// TwinCAT 3 PLC project MasterArmControl
// ProgramVersion: 3.1.4024.0
// libraries:
//   Tc2_Math, * (Beckhoff Automation GmbH)
//   Tc2_Standard, * (Beckhoff Automation GmbH)
//   Tc2_System, * (Beckhoff Automation GmbH)
//   Tc2_Utilities, * (Beckhoff Automation GmbH)
//   Tc3_Module, * (Beckhoff Automation GmbH)
// project tree:
//   AgiMaths/ DHTrans.TcPOU, sign.TcPOU, addVec7.TcPOU (not stored), multiNumVec3.TcPOU, multiNumVec7.TcPOU, normVec3.TcPOU, normVec7.TcPOU, subVec7.TcPOU (not stored), subVec3.TcPOU (not stored), addVec3.TcPOU (not stored), atan2.TcPOU (not stored), cot.TcPOU (not stored), mat3Mat3.TcPOU (not stored), mat3Vec3.TcPOU (not stored), mat67Vec7.TcPOU (not stored), rotZ.TcPOU (not stored), rotY.TcPOU (not stored), rotX.TcPOU (not stored), transform.TcPOU (not stored)
//   DUTs/Structure/Communication/ ST_MasterDynaData.TcDUT, ST_UIData.TcDUT, ST_CartStatus.TcDUT, ST_MasterStatus.TcDUT, ST_MasterJointData.TcDUT, ST_MotorInputs.TcDUT (not stored), ST_MotorOutputs.TcDUT (not stored), ST_SlaveStatus.TcDUT, ST_SlaveJointData.TcDUT, ST_SafetyData.TcDUT (not stored)
//   DUTs/Structure/ ST_ArmCtrlCmds.TcDUT, ST_MasterInputDataPool.TcDUT, ST_Frame.TcDUT, ST_InstruStatus.TcDUT
//   DUTs/Type/ Mat37.TcDUT (not stored), Mat4d.TcDUT (not stored), Mat5d.TcDUT (not stored), Mat67.TcDUT, Mat6d.TcDUT, Mat76.TcDUT, Mat7d.TcDUT, Vec4d.TcDUT (not stored), Mat3d.TcDUT, Vec3d.TcDUT, Vec6d.TcDUT, Vec7d.TcDUT (not stored), Vec7i.TcDUT (not stored)
//   FBs_BasicControllers/ FB_RedunJntControl.TcPOU (not stored), FB_PID.TcPOU
//   DUTs/Enum/ E_DriverCtrlWord.TcDUT (not stored), E_DriverOPMode.TcDUT (not stored), E_DriverStatusWord.TcDUT, E_InstrumentType.TcDUT (not stored), E_MasterArmState.TcDUT (not stored), E_MatchedSlaveArmIdx.TcDUT (not stored), E_SlaveArmState.TcDUT
//   FBs_RobotDynamics/ FB_MasterDynamic.TcPOU, FB_MasterGravity.TcPOU
//   FBs_StateControllers/ FB_ArmClutch.TcPOU, FB_ArmEndoscope.TcPOU, FB_ArmCart.TcPOU, FB_ArmMatching.TcPOU, FB_ArmHome.TcPOU, FB_ArmError.TcPOU, FB_ArmReady.TcPOU, FB_ArmMasterSlave.TcPOU, FB_ArmInit.TcPOU, FB_ArmStandBy.TcPOU, FB_MasterArmCtrlBase.TcPOU, I_MasterArmCtrl.TcIO
//   FBs_TrajectoryPlanning/ FB_BasicDoubleS.TcPOU, FB_trajBase.TcPOU (not stored), FB_TrajMoveJ.TcPOU, linear_trajectory_with_quintic_polynomial_blends.TcPOU, quintic_spline_curve.TcPOU, Quintic_spline_curve_factor.TcPOU, TrapezoIDal_velocity_trajectory.TcPOU
//   FBs_TrajectoryPlanning/OTG/ FB_secOrdTrajFilter.TcPOU (not stored), FB_thirdOrdTrajFilter.TcPOU
//   FBs_Filters/ FB_LowPassFilter.TcPOU (not stored)
//   GVLs/ GVLs_ArmDynamics.TcGVL (not stored), GVL_ArmKinematic.TcGVL (not stored), GVL_CartParameters.TcGVL (not stored), GVL_ControlParameters.TcGVL, GVL_JointEncoderCaliData.TcGVL, GVL_MathDefine.TcGVL, GVL_MotorParameters.TcGVL, GVL_SafetyParameters.TcGVL (not stored), GVL_SystemParameters.TcGVL
//   FBs_Robots/ FB_Joint.TcPOU, FB_MasterArm.TcPOU, FB_MasterRobot.TcPOU
//   MatrixLib/ cross.TcPOU, Det5.TcPOU, Det6.TcPOU, Det7.TcPOU, invMat6Old.TcPOU, invMat7.TcPOU, invMat6.TcPOU, Mat3T.TcPOU, vecSelfMultiNum.TcPOU, matMultiVec.TcPOU, matMultiply.TcPOU, matMultiNum.TcPOU, matSelfSub.TcPOU, matAdd.TcPOU, matSelfAdd.TcPOU (not stored), matTranspose.TcPOU, matSub.TcPOU (not stored)
//   / TaskArmControl.TcTTO, TaskDynamic.TcTTO
//   Mains/ MasterArmControl.TcPOU, RobotDynamics.TcPOU
// real-time tasks:
//   TASK TaskArmControl: cycle T#1ms, priority 20, ADS port 350
//   TASK TaskDynamic: cycle T#1ms, priority 1, ADS port 351
// I/O:
//   DEVICE Device 3 (EtherCAT) (disabled), AmsNetId 169.254.206.98.4.1
//     Box 26 (AX58200_MotorControl) [AX58200_MotorControl2021.9.13]
//     Box 27 (EL6695-0002) [EL6695 EtherCAT Bridge terminal (Secondary)]
//   DEVICE LeftArm (EtherCAT), AmsNetId 169.254.206.98.3.1
//     Joint1 (AX58200_MotorControl) [AX58200_MotorControl_1axis]
//     Joint2 (AX58200_MotorControl) [AX58200_MotorControl_1axis]
//     Joint3 (AX58200_MotorControl) [AX58200_MotorControl_1axis]
//     Joint4 (AX58200_MotorControl) [AX58200_MotorControl_1axis]
//     Joint5 (AX58200_MotorControl) [AX58200_MotorControl_1axis]
//     Joint6 (AX58200_MotorControl) [AX58200_MotorControl_1axis]
//     Joint7 (AX58200_MotorControl) [AX58200_MotorControl_1axis]
//   DEVICE RightArm (EtherCAT), AmsNetId 169.254.206.98.7.1
//     Term 1 (EK1100) [EK1100 EtherCAT Coupler (2A E-Bus)]
//       Term 2 (EL6070) [EL6070 1Ch. Licensing-Terminal]
//       Term 3 (EL1008) [EL1008 8Ch. Dig. Input 24V, 3ms]
//       Term 4 (EL1008) [EL1008 8Ch. Dig. Input 24V, 3ms]
//       Term 5 (EL1008) [EL1008 8Ch. Dig. Input 24V, 3ms]
//       Term 6 (EL2008-0015) [EL2008-0015 8K. Dig. Ausgang 24V DC, 0.35A, nicht kurzschlussfest]
//       Term 7 (EK1122) [EK1122 2 port EtherCAT junction]
//         Box 8 (AX58200_MotorControl) [AX58200_MotorControl_1axis]
//         Box 9 (AX58200_MotorControl) [AX58200_MotorControl_1axis]
//         Box 10 (AX58200_MotorControl) [AX58200_MotorControl_1axis]
//         Box 11 (AX58200_MotorControl) [AX58200_MotorControl_1axis]
//     Joint1 (AX58200_MotorControl) [AX58200_MotorControl_1axis]
//     Joint2 (AX58200_MotorControl) [AX58200_MotorControl_1axis]
//     Joint3 (AX58200_MotorControl) [AX58200_MotorControl_1axis]
//     Joint4 (AX58200_MotorControl) [AX58200_MotorControl_1axis]
//     Joint5 (AX58200_MotorControl) [AX58200_MotorControl_1axis]
//     Joint6 (AX58200_MotorControl) [AX58200_MotorControl_1axis]
//     Joint7 (AX58200_MotorControl) [AX58200_MotorControl_1axis]
// variable links:
//   MasterArmControl/MasterArmControl Instance <-> LeftArm (EtherCAT)/Joint1 (AX58200_MotorControl)
//     TaskArmControl Inputs/MasterArmControl.m_masterRobot.m_masterArms[1].m_joints[1].m_motorInputs/m_current <-> TxPdoMappingCspCsv/Torque actual value
//     TaskArmControl Inputs/MasterArmControl.m_masterRobot.m_masterArms[1].m_joints[1].m_motorInputs/m_driverError <-> TxPdoMappingCspCsv/digital input
//     TaskArmControl Inputs/MasterArmControl.m_masterRobot.m_masterArms[1].m_joints[1].m_motorInputs/m_linkEncoder <-> TxPdoMappingCspCsv/ENC2
//     TaskArmControl Inputs/MasterArmControl.m_masterRobot.m_masterArms[1].m_joints[1].m_motorInputs/m_motorEncoder <-> TxPdoMappingCspCsv/Position actual value
//     TaskArmControl Inputs/MasterArmControl.m_masterRobot.m_masterArms[1].m_joints[1].m_motorInputs/m_statusWord <-> TxPdoMappingCspCsv/Statusword
//     TaskArmControl Outputs/MasterArmControl.m_masterRobot.m_masterArms[1].m_joints[1].m_motorOutputs/m_cmdCurrent <-> RxPdoMappingCspCsv/Target torque
//     TaskArmControl Outputs/MasterArmControl.m_masterRobot.m_masterArms[1].m_joints[1].m_motorOutputs/m_cmdMotorEncoder <-> RxPdoMappingCspCsv/Target position
//     TaskArmControl Outputs/MasterArmControl.m_masterRobot.m_masterArms[1].m_joints[1].m_motorOutputs/m_controlWord <-> RxPdoMappingCspCsv/Controlword
//     TaskArmControl Outputs/MasterArmControl.m_masterRobot.m_masterArms[1].m_joints[1].m_motorOutputs/m_opMode <-> RxPdoMappingCspCsv/Modes of operation
//   MasterArmControl/MasterArmControl Instance <-> LeftArm (EtherCAT)/Joint2 (AX58200_MotorControl)
//     TaskArmControl Inputs/MasterArmControl.m_masterRobot.m_masterArms[1].m_joints[2].m_motorInputs/m_current <-> TxPdoMappingCspCsv/Torque actual value
//     TaskArmControl Inputs/MasterArmControl.m_masterRobot.m_masterArms[1].m_joints[2].m_motorInputs/m_driverError <-> TxPdoMappingCspCsv/digital input
//     TaskArmControl Inputs/MasterArmControl.m_masterRobot.m_masterArms[1].m_joints[2].m_motorInputs/m_linkEncoder <-> TxPdoMappingCspCsv/ENC2
//     TaskArmControl Inputs/MasterArmControl.m_masterRobot.m_masterArms[1].m_joints[2].m_motorInputs/m_motorEncoder <-> TxPdoMappingCspCsv/Position actual value
//     TaskArmControl Inputs/MasterArmControl.m_masterRobot.m_masterArms[1].m_joints[2].m_motorInputs/m_statusWord <-> TxPdoMappingCspCsv/Statusword
//     TaskArmControl Outputs/MasterArmControl.m_masterRobot.m_masterArms[1].m_joints[2].m_motorOutputs/m_cmdCurrent <-> RxPdoMappingCspCsv/Target torque
//     TaskArmControl Outputs/MasterArmControl.m_masterRobot.m_masterArms[1].m_joints[2].m_motorOutputs/m_cmdMotorEncoder <-> RxPdoMappingCspCsv/Target position
//     TaskArmControl Outputs/MasterArmControl.m_masterRobot.m_masterArms[1].m_joints[2].m_motorOutputs/m_controlWord <-> RxPdoMappingCspCsv/Controlword
//     TaskArmControl Outputs/MasterArmControl.m_masterRobot.m_masterArms[1].m_joints[2].m_motorOutputs/m_opMode <-> RxPdoMappingCspCsv/Modes of operation
//   MasterArmControl/MasterArmControl Instance <-> LeftArm (EtherCAT)/Joint3 (AX58200_MotorControl)
//     TaskArmControl Inputs/MasterArmControl.m_masterRobot.m_masterArms[1].m_joints[3].m_motorInputs/m_current <-> TxPdoMappingCspCsv/Torque actual value
//     TaskArmControl Inputs/MasterArmControl.m_masterRobot.m_masterArms[1].m_joints[3].m_motorInputs/m_driverError <-> TxPdoMappingCspCsv/digital input
//     TaskArmControl Inputs/MasterArmControl.m_masterRobot.m_masterArms[1].m_joints[3].m_motorInputs/m_linkEncoder <-> TxPdoMappingCspCsv/ENC2
//     TaskArmControl Inputs/MasterArmControl.m_masterRobot.m_masterArms[1].m_joints[3].m_motorInputs/m_motorEncoder <-> TxPdoMappingCspCsv/Position actual value
//     TaskArmControl Inputs/MasterArmControl.m_masterRobot.m_masterArms[1].m_joints[3].m_motorInputs/m_statusWord <-> TxPdoMappingCspCsv/Statusword
//     TaskArmControl Outputs/MasterArmControl.m_masterRobot.m_masterArms[1].m_joints[3].m_motorOutputs/m_cmdCurrent <-> RxPdoMappingCspCsv/Target torque
//     TaskArmControl Outputs/MasterArmControl.m_masterRobot.m_masterArms[1].m_joints[3].m_motorOutputs/m_cmdMotorEncoder <-> RxPdoMappingCspCsv/Target position
//     TaskArmControl Outputs/MasterArmControl.m_masterRobot.m_masterArms[1].m_joints[3].m_motorOutputs/m_controlWord <-> RxPdoMappingCspCsv/Controlword
//     TaskArmControl Outputs/MasterArmControl.m_masterRobot.m_masterArms[1].m_joints[3].m_motorOutputs/m_opMode <-> RxPdoMappingCspCsv/Modes of operation
//   MasterArmControl/MasterArmControl Instance <-> LeftArm (EtherCAT)/Joint4 (AX58200_MotorControl)
//     TaskArmControl Inputs/MasterArmControl.m_masterRobot.m_masterArms[1].m_joints[4].m_motorInputs/m_current <-> TxPdoMappingCspCsv/Torque actual value
//     TaskArmControl Inputs/MasterArmControl.m_masterRobot.m_masterArms[1].m_joints[4].m_motorInputs/m_driverError <-> TxPdoMappingCspCsv/digital input
//     TaskArmControl Inputs/MasterArmControl.m_masterRobot.m_masterArms[1].m_joints[4].m_motorInputs/m_motorEncoder <-> TxPdoMappingCspCsv/Position actual value
//     TaskArmControl Inputs/MasterArmControl.m_masterRobot.m_masterArms[1].m_joints[4].m_motorInputs/m_statusWord <-> TxPdoMappingCspCsv/Statusword
//     TaskArmControl Outputs/MasterArmControl.m_masterRobot.m_masterArms[1].m_joints[4].m_motorOutputs/m_cmdCurrent <-> RxPdoMappingCspCsv/Target torque
//     TaskArmControl Outputs/MasterArmControl.m_masterRobot.m_masterArms[1].m_joints[4].m_motorOutputs/m_cmdMotorEncoder <-> RxPdoMappingCspCsv/Target position
//     TaskArmControl Outputs/MasterArmControl.m_masterRobot.m_masterArms[1].m_joints[4].m_motorOutputs/m_controlWord <-> RxPdoMappingCspCsv/Controlword
//     TaskArmControl Outputs/MasterArmControl.m_masterRobot.m_masterArms[1].m_joints[4].m_motorOutputs/m_opMode <-> RxPdoMappingCspCsv/Modes of operation
//   MasterArmControl/MasterArmControl Instance <-> LeftArm (EtherCAT)/Joint5 (AX58200_MotorControl)
//     TaskArmControl Inputs/MasterArmControl.m_masterRobot.m_masterArms[1].m_joints[4].m_motorInputs/m_linkEncoder <-> TxPdoMappingCspCsv/Velocity actual value
//     TaskArmControl Inputs/MasterArmControl.m_masterRobot.m_masterArms[1].m_joints[5].m_motorInputs/m_current <-> TxPdoMappingCspCsv/Torque actual value
//     TaskArmControl Inputs/MasterArmControl.m_masterRobot.m_masterArms[1].m_joints[5].m_motorInputs/m_driverError <-> TxPdoMappingCspCsv/digital input
//     TaskArmControl Inputs/MasterArmControl.m_masterRobot.m_masterArms[1].m_joints[5].m_motorInputs/m_linkEncoder <-> TxPdoMappingCspCsv/ENC2
//     TaskArmControl Inputs/MasterArmControl.m_masterRobot.m_masterArms[1].m_joints[5].m_motorInputs/m_motorEncoder <-> TxPdoMappingCspCsv/Position actual value
//     TaskArmControl Inputs/MasterArmControl.m_masterRobot.m_masterArms[1].m_joints[5].m_motorInputs/m_statusWord <-> TxPdoMappingCspCsv/Statusword
//     TaskArmControl Outputs/MasterArmControl.m_masterRobot.m_masterArms[1].m_joints[5].m_motorOutputs/m_cmdCurrent <-> RxPdoMappingCspCsv/Target torque
//     TaskArmControl Outputs/MasterArmControl.m_masterRobot.m_masterArms[1].m_joints[5].m_motorOutputs/m_cmdMotorEncoder <-> RxPdoMappingCspCsv/Target position
//     TaskArmControl Outputs/MasterArmControl.m_masterRobot.m_masterArms[1].m_joints[5].m_motorOutputs/m_controlWord <-> RxPdoMappingCspCsv/Controlword
//     TaskArmControl Outputs/MasterArmControl.m_masterRobot.m_masterArms[1].m_joints[5].m_motorOutputs/m_opMode <-> RxPdoMappingCspCsv/Modes of operation
//   MasterArmControl/MasterArmControl Instance <-> LeftArm (EtherCAT)/Joint6 (AX58200_MotorControl)
//     TaskArmControl Inputs/MasterArmControl.m_masterRobot.m_masterArms[1].m_joints[6].m_motorInputs/m_current <-> TxPdoMappingCspCsv/Torque actual value
//     TaskArmControl Inputs/MasterArmControl.m_masterRobot.m_masterArms[1].m_joints[6].m_motorInputs/m_driverError <-> TxPdoMappingCspCsv/digital input
//     TaskArmControl Inputs/MasterArmControl.m_masterRobot.m_masterArms[1].m_joints[6].m_motorInputs/m_linkEncoder <-> TxPdoMappingCspCsv/ENC2
//     TaskArmControl Inputs/MasterArmControl.m_masterRobot.m_masterArms[1].m_joints[6].m_motorInputs/m_motorEncoder <-> TxPdoMappingCspCsv/Position actual value
//     TaskArmControl Inputs/MasterArmControl.m_masterRobot.m_masterArms[1].m_joints[6].m_motorInputs/m_statusWord <-> TxPdoMappingCspCsv/Statusword
//     TaskArmControl Outputs/MasterArmControl.m_masterRobot.m_masterArms[1].m_joints[6].m_motorOutputs/m_cmdCurrent <-> RxPdoMappingCspCsv/Target torque
//     TaskArmControl Outputs/MasterArmControl.m_masterRobot.m_masterArms[1].m_joints[6].m_motorOutputs/m_cmdMotorEncoder <-> RxPdoMappingCspCsv/Target position
//     TaskArmControl Outputs/MasterArmControl.m_masterRobot.m_masterArms[1].m_joints[6].m_motorOutputs/m_controlWord <-> RxPdoMappingCspCsv/Controlword
//     TaskArmControl Outputs/MasterArmControl.m_masterRobot.m_masterArms[1].m_joints[6].m_motorOutputs/m_opMode <-> RxPdoMappingCspCsv/Modes of operation
//   MasterArmControl/MasterArmControl Instance <-> LeftArm (EtherCAT)/Joint7 (AX58200_MotorControl)
//     TaskArmControl Inputs/MasterArmControl.m_masterRobot.m_masterArms[1].m_gripHallSensorValue <-> TxPdoMappingCspCsv/analog input
//     TaskArmControl Inputs/MasterArmControl.m_masterRobot.m_masterArms[1].m_joints[7].m_motorInputs/m_current <-> TxPdoMappingCspCsv/Torque actual value
//     TaskArmControl Inputs/MasterArmControl.m_masterRobot.m_masterArms[1].m_joints[7].m_motorInputs/m_driverError <-> TxPdoMappingCspCsv/digital input
//     TaskArmControl Inputs/MasterArmControl.m_masterRobot.m_masterArms[1].m_joints[7].m_motorInputs/m_linkEncoder <-> TxPdoMappingCspCsv/ENC2
//     TaskArmControl Inputs/MasterArmControl.m_masterRobot.m_masterArms[1].m_joints[7].m_motorInputs/m_motorEncoder <-> TxPdoMappingCspCsv/Position actual value
//     TaskArmControl Inputs/MasterArmControl.m_masterRobot.m_masterArms[1].m_joints[7].m_motorInputs/m_statusWord <-> TxPdoMappingCspCsv/Statusword
//     TaskArmControl Outputs/MasterArmControl.m_masterRobot.m_masterArms[1].m_joints[7].m_motorOutputs/m_cmdCurrent <-> RxPdoMappingCspCsv/Target torque
//     TaskArmControl Outputs/MasterArmControl.m_masterRobot.m_masterArms[1].m_joints[7].m_motorOutputs/m_cmdMotorEncoder <-> RxPdoMappingCspCsv/Target position
//     TaskArmControl Outputs/MasterArmControl.m_masterRobot.m_masterArms[1].m_joints[7].m_motorOutputs/m_controlWord <-> RxPdoMappingCspCsv/Controlword
//     TaskArmControl Outputs/MasterArmControl.m_masterRobot.m_masterArms[1].m_joints[7].m_motorOutputs/m_opMode <-> RxPdoMappingCspCsv/Modes of operation
//   MasterArmControl/MasterArmControl Instance <-> RightArm (EtherCAT)/Joint1 (AX58200_MotorControl)
//     TaskArmControl Inputs/MasterArmControl.m_masterRobot.m_masterArms[2].m_joints[1].m_motorInputs/m_current <-> TxPdoMappingCspCsv/Torque actual value
//     TaskArmControl Inputs/MasterArmControl.m_masterRobot.m_masterArms[2].m_joints[1].m_motorInputs/m_driverError <-> TxPdoMappingCspCsv/digital input
//     TaskArmControl Inputs/MasterArmControl.m_masterRobot.m_masterArms[2].m_joints[1].m_motorInputs/m_linkEncoder <-> TxPdoMappingCspCsv/ENC2
//     TaskArmControl Inputs/MasterArmControl.m_masterRobot.m_masterArms[2].m_joints[1].m_motorInputs/m_motorEncoder <-> TxPdoMappingCspCsv/Position actual value
//     TaskArmControl Inputs/MasterArmControl.m_masterRobot.m_masterArms[2].m_joints[1].m_motorInputs/m_statusWord <-> TxPdoMappingCspCsv/Statusword
//     TaskArmControl Outputs/MasterArmControl.m_masterRobot.m_masterArms[2].m_joints[1].m_motorOutputs/m_cmdCurrent <-> RxPdoMappingCspCsv/Target torque
//     TaskArmControl Outputs/MasterArmControl.m_masterRobot.m_masterArms[2].m_joints[1].m_motorOutputs/m_cmdMotorEncoder <-> RxPdoMappingCspCsv/Target position
//     TaskArmControl Outputs/MasterArmControl.m_masterRobot.m_masterArms[2].m_joints[1].m_motorOutputs/m_controlWord <-> RxPdoMappingCspCsv/Controlword
//     TaskArmControl Outputs/MasterArmControl.m_masterRobot.m_masterArms[2].m_joints[1].m_motorOutputs/m_opMode <-> RxPdoMappingCspCsv/Modes of operation
//   MasterArmControl/MasterArmControl Instance <-> RightArm (EtherCAT)/Joint2 (AX58200_MotorControl)
//     TaskArmControl Inputs/MasterArmControl.m_masterRobot.m_masterArms[2].m_joints[2].m_motorInputs/m_current <-> TxPdoMappingCspCsv/Torque actual value
//     TaskArmControl Inputs/MasterArmControl.m_masterRobot.m_masterArms[2].m_joints[2].m_motorInputs/m_driverError <-> TxPdoMappingCspCsv/digital input
//     TaskArmControl Inputs/MasterArmControl.m_masterRobot.m_masterArms[2].m_joints[2].m_motorInputs/m_linkEncoder <-> TxPdoMappingCspCsv/ENC2
//     TaskArmControl Inputs/MasterArmControl.m_masterRobot.m_masterArms[2].m_joints[2].m_motorInputs/m_motorEncoder <-> TxPdoMappingCspCsv/Position actual value
//     TaskArmControl Inputs/MasterArmControl.m_masterRobot.m_masterArms[2].m_joints[2].m_motorInputs/m_statusWord <-> TxPdoMappingCspCsv/Statusword
//     TaskArmControl Outputs/MasterArmControl.m_masterRobot.m_masterArms[2].m_joints[2].m_motorOutputs/m_cmdCurrent <-> RxPdoMappingCspCsv/Target torque
//     TaskArmControl Outputs/MasterArmControl.m_masterRobot.m_masterArms[2].m_joints[2].m_motorOutputs/m_cmdMotorEncoder <-> RxPdoMappingCspCsv/Target position
//     TaskArmControl Outputs/MasterArmControl.m_masterRobot.m_masterArms[2].m_joints[2].m_motorOutputs/m_controlWord <-> RxPdoMappingCspCsv/Controlword
//     TaskArmControl Outputs/MasterArmControl.m_masterRobot.m_masterArms[2].m_joints[2].m_motorOutputs/m_opMode <-> RxPdoMappingCspCsv/Modes of operation
//   MasterArmControl/MasterArmControl Instance <-> RightArm (EtherCAT)/Joint3 (AX58200_MotorControl)
//     TaskArmControl Inputs/MasterArmControl.m_masterRobot.m_masterArms[2].m_joints[3].m_motorInputs/m_current <-> TxPdoMappingCspCsv/Torque actual value
//     TaskArmControl Inputs/MasterArmControl.m_masterRobot.m_masterArms[2].m_joints[3].m_motorInputs/m_driverError <-> TxPdoMappingCspCsv/digital input
//     TaskArmControl Inputs/MasterArmControl.m_masterRobot.m_masterArms[2].m_joints[3].m_motorInputs/m_linkEncoder <-> TxPdoMappingCspCsv/ENC2
//     TaskArmControl Inputs/MasterArmControl.m_masterRobot.m_masterArms[2].m_joints[3].m_motorInputs/m_motorEncoder <-> TxPdoMappingCspCsv/Position actual value
//     TaskArmControl Inputs/MasterArmControl.m_masterRobot.m_masterArms[2].m_joints[3].m_motorInputs/m_statusWord <-> TxPdoMappingCspCsv/Statusword
//     TaskArmControl Outputs/MasterArmControl.m_masterRobot.m_masterArms[2].m_joints[3].m_motorOutputs/m_cmdCurrent <-> RxPdoMappingCspCsv/Target torque
//     TaskArmControl Outputs/MasterArmControl.m_masterRobot.m_masterArms[2].m_joints[3].m_motorOutputs/m_cmdMotorEncoder <-> RxPdoMappingCspCsv/Target position
//     TaskArmControl Outputs/MasterArmControl.m_masterRobot.m_masterArms[2].m_joints[3].m_motorOutputs/m_controlWord <-> RxPdoMappingCspCsv/Controlword
//     TaskArmControl Outputs/MasterArmControl.m_masterRobot.m_masterArms[2].m_joints[3].m_motorOutputs/m_opMode <-> RxPdoMappingCspCsv/Modes of operation
//   MasterArmControl/MasterArmControl Instance <-> RightArm (EtherCAT)/Joint4 (AX58200_MotorControl)
//     TaskArmControl Inputs/MasterArmControl.m_masterRobot.m_masterArms[2].m_joints[4].m_motorInputs/m_current <-> TxPdoMappingCspCsv/Torque actual value
//     TaskArmControl Inputs/MasterArmControl.m_masterRobot.m_masterArms[2].m_joints[4].m_motorInputs/m_driverError <-> TxPdoMappingCspCsv/digital input
//     TaskArmControl Inputs/MasterArmControl.m_masterRobot.m_masterArms[2].m_joints[4].m_motorInputs/m_motorEncoder <-> TxPdoMappingCspCsv/Position actual value
//     TaskArmControl Inputs/MasterArmControl.m_masterRobot.m_masterArms[2].m_joints[4].m_motorInputs/m_statusWord <-> TxPdoMappingCspCsv/Statusword
//     TaskArmControl Outputs/MasterArmControl.m_masterRobot.m_masterArms[2].m_joints[4].m_motorOutputs/m_cmdCurrent <-> RxPdoMappingCspCsv/Target torque
//     TaskArmControl Outputs/MasterArmControl.m_masterRobot.m_masterArms[2].m_joints[4].m_motorOutputs/m_cmdMotorEncoder <-> RxPdoMappingCspCsv/Target position
//     TaskArmControl Outputs/MasterArmControl.m_masterRobot.m_masterArms[2].m_joints[4].m_motorOutputs/m_controlWord <-> RxPdoMappingCspCsv/Controlword
//     TaskArmControl Outputs/MasterArmControl.m_masterRobot.m_masterArms[2].m_joints[4].m_motorOutputs/m_opMode <-> RxPdoMappingCspCsv/Modes of operation
//   MasterArmControl/MasterArmControl Instance <-> RightArm (EtherCAT)/Joint5 (AX58200_MotorControl)
//     TaskArmControl Inputs/MasterArmControl.m_masterRobot.m_masterArms[2].m_joints[4].m_motorInputs/m_linkEncoder <-> TxPdoMappingCspCsv/Velocity actual value
//     TaskArmControl Inputs/MasterArmControl.m_masterRobot.m_masterArms[2].m_joints[5].m_motorInputs/m_current <-> TxPdoMappingCspCsv/Torque actual value
//     TaskArmControl Inputs/MasterArmControl.m_masterRobot.m_masterArms[2].m_joints[5].m_motorInputs/m_driverError <-> TxPdoMappingCspCsv/digital input
//     TaskArmControl Inputs/MasterArmControl.m_masterRobot.m_masterArms[2].m_joints[5].m_motorInputs/m_linkEncoder <-> TxPdoMappingCspCsv/ENC2
//     TaskArmControl Inputs/MasterArmControl.m_masterRobot.m_masterArms[2].m_joints[5].m_motorInputs/m_motorEncoder <-> TxPdoMappingCspCsv/Position actual value
//     TaskArmControl Inputs/MasterArmControl.m_masterRobot.m_masterArms[2].m_joints[5].m_motorInputs/m_statusWord <-> TxPdoMappingCspCsv/Statusword
//     TaskArmControl Outputs/MasterArmControl.m_masterRobot.m_masterArms[2].m_joints[5].m_motorOutputs/m_cmdCurrent <-> RxPdoMappingCspCsv/Target torque
//     TaskArmControl Outputs/MasterArmControl.m_masterRobot.m_masterArms[2].m_joints[5].m_motorOutputs/m_cmdMotorEncoder <-> RxPdoMappingCspCsv/Target position
//     TaskArmControl Outputs/MasterArmControl.m_masterRobot.m_masterArms[2].m_joints[5].m_motorOutputs/m_controlWord <-> RxPdoMappingCspCsv/Controlword
//     TaskArmControl Outputs/MasterArmControl.m_masterRobot.m_masterArms[2].m_joints[5].m_motorOutputs/m_opMode <-> RxPdoMappingCspCsv/Modes of operation
//   MasterArmControl/MasterArmControl Instance <-> RightArm (EtherCAT)/Joint6 (AX58200_MotorControl)
//     TaskArmControl Inputs/MasterArmControl.m_masterRobot.m_masterArms[2].m_joints[6].m_motorInputs/m_current <-> TxPdoMappingCspCsv/Torque actual value
//     TaskArmControl Inputs/MasterArmControl.m_masterRobot.m_masterArms[2].m_joints[6].m_motorInputs/m_driverError <-> TxPdoMappingCspCsv/digital input
//     TaskArmControl Inputs/MasterArmControl.m_masterRobot.m_masterArms[2].m_joints[6].m_motorInputs/m_linkEncoder <-> TxPdoMappingCspCsv/ENC2
//     TaskArmControl Inputs/MasterArmControl.m_masterRobot.m_masterArms[2].m_joints[6].m_motorInputs/m_motorEncoder <-> TxPdoMappingCspCsv/Position actual value
//     TaskArmControl Inputs/MasterArmControl.m_masterRobot.m_masterArms[2].m_joints[6].m_motorInputs/m_statusWord <-> TxPdoMappingCspCsv/Statusword
//     TaskArmControl Outputs/MasterArmControl.m_masterRobot.m_masterArms[2].m_joints[6].m_motorOutputs/m_cmdCurrent <-> RxPdoMappingCspCsv/Target torque
//     TaskArmControl Outputs/MasterArmControl.m_masterRobot.m_masterArms[2].m_joints[6].m_motorOutputs/m_cmdMotorEncoder <-> RxPdoMappingCspCsv/Target position
//     TaskArmControl Outputs/MasterArmControl.m_masterRobot.m_masterArms[2].m_joints[6].m_motorOutputs/m_controlWord <-> RxPdoMappingCspCsv/Controlword
//     TaskArmControl Outputs/MasterArmControl.m_masterRobot.m_masterArms[2].m_joints[6].m_motorOutputs/m_opMode <-> RxPdoMappingCspCsv/Modes of operation
//   MasterArmControl/MasterArmControl Instance <-> RightArm (EtherCAT)/Joint7 (AX58200_MotorControl)
//     TaskArmControl Inputs/MasterArmControl.m_masterRobot.m_masterArms[2].m_gripHallSensorValue <-> TxPdoMappingCspCsv/analog input
//     TaskArmControl Inputs/MasterArmControl.m_masterRobot.m_masterArms[2].m_joints[7].m_motorInputs/m_current <-> TxPdoMappingCspCsv/Torque actual value
//     TaskArmControl Inputs/MasterArmControl.m_masterRobot.m_masterArms[2].m_joints[7].m_motorInputs/m_driverError <-> TxPdoMappingCspCsv/digital input
//     TaskArmControl Inputs/MasterArmControl.m_masterRobot.m_masterArms[2].m_joints[7].m_motorInputs/m_linkEncoder <-> TxPdoMappingCspCsv/ENC2
//     TaskArmControl Inputs/MasterArmControl.m_masterRobot.m_masterArms[2].m_joints[7].m_motorInputs/m_motorEncoder <-> TxPdoMappingCspCsv/Position actual value
//     TaskArmControl Inputs/MasterArmControl.m_masterRobot.m_masterArms[2].m_joints[7].m_motorInputs/m_statusWord <-> TxPdoMappingCspCsv/Statusword
//     TaskArmControl Outputs/MasterArmControl.m_masterRobot.m_masterArms[2].m_joints[7].m_motorOutputs/m_cmdCurrent <-> RxPdoMappingCspCsv/Target torque
//     TaskArmControl Outputs/MasterArmControl.m_masterRobot.m_masterArms[2].m_joints[7].m_motorOutputs/m_cmdMotorEncoder <-> RxPdoMappingCspCsv/Target position
//     TaskArmControl Outputs/MasterArmControl.m_masterRobot.m_masterArms[2].m_joints[7].m_motorOutputs/m_controlWord <-> RxPdoMappingCspCsv/Controlword
//     TaskArmControl Outputs/MasterArmControl.m_masterRobot.m_masterArms[2].m_joints[7].m_motorOutputs/m_opMode <-> RxPdoMappingCspCsv/Modes of operation
//   MasterArmControl/MasterArmControl Instance <-> MasterArmControl/MasterArmControl Instance
//     TaskArmControl Inputs/MasterArmControl.m_masterInputDataPool.m_masterDynaData <-> TaskDynamic Outputs/RobotDynamics.m_masterDynaData
//     TaskDynamic Inputs/RobotDynamics.m_masterJointsData <-> TaskArmControl Outputs/MasterArmControl.m_masterJointsData

CONFIGURATION MasterArmControl
    RESOURCE PLC ON TwinCAT3
        TASK TaskArmControl(INTERVAL := T#1ms, PRIORITY := 20);
        TASK TaskDynamic(INTERVAL := T#1ms, PRIORITY := 1);
        PROGRAM MasterArmControl WITH TaskArmControl : MasterArmControl;
        PROGRAM RobotDynamics WITH TaskDynamic : RobotDynamics;
    END_RESOURCE
END_CONFIGURATION

// ---- DUTs/Structure/Communication/ST_MasterDynaData.TcDUT
TYPE ST_MasterDynaData :
STRUCT
	// mass matrix in joint space
	m_massMat :ARRAY[1..g_mArmNum] OF Mat7d;
	
	// mass matrix in cartesian space
	m_lambda :ARRAY[1..g_mArmNum] OF Mat6d;
	
	// dynamic nullspace
	m_dynaNullspace :ARRAY[1..g_mArmNum] OF Mat7d;
	
	// gravity
	m_gravity :ARRAY[1..g_mArmNum] OF Vec7d;
END_STRUCT
END_TYPE

// ---- DUTs/Structure/Communication/ST_UIData.TcDUT
// Output from UI controller
// Input to master arm control task and cart control task  
TYPE ST_UIData :
STRUCT
	m_motionScale:LREAL := 1.0;
	m_faultClearFlag:BOOL := FALSE;
END_STRUCT
END_TYPE

// ---- DUTs/Structure/Communication/ST_CartStatus.TcDUT
// Output from cart control task
// Input to master arm control task  
TYPE ST_CartStatus :
STRUCT
	m_monitorAngle:LREAL := 0.0;
	m_armSwitch:BOOL := FALSE;
	m_clutchSwitch:BOOL := FALSE;
	m_endoscopeSwitch:BOOL := FALSE;
	m_instrumentPowerSwitch:BOOL := FALSE;
	m_monitorAdjustSwitch:BOOL := FALSE;
	m_tableAdjustSwitch:BOOL := FALSE;
END_STRUCT
END_TYPE

// ---- DUTs/Structure/Communication/ST_MasterStatus.TcDUT
// Output from master arm control task, including arm status and cartesian data
// Input to safety task and Slave controller
TYPE ST_MasterStatus :
STRUCT
	// linear motion scale
	m_motionScale : LREAL;
	
	// state machine
	m_armState:ARRAY[1..g_mArmNum] OF E_masterArmState;
	
	// index(0 to 4) of slave arm which is tele-linked to master arm
	m_teleSlaveArmIdx :ARRAY[1..g_mArmNum] OF E_MatchedSlaveArmIdx;
	
	// grip angle
	m_gripAngle:ARRAY[1..g_mArmNum] OF LREAL;
	
	// command arm pose in monitor
	m_cmdArmPose :ARRAY[1..g_mArmNum] OF ST_Frame;
	
	// current arm pose in monitor
	m_curArmPose:ARRAY[1..g_mArmNum] OF ST_Frame;
	
	// command arm twist[linear velocity; angular veloicty] in monitor
	m_cmdArmTwist:ARRAY[1..g_mArmNum] OF Vec6d;
	
	// current arm twist[linear velocity; angular veloicty] in monitor
	m_curArmTwist:ARRAY[1..g_mArmNum] OF Vec6d;
	
END_STRUCT
END_TYPE

// ---- DUTs/Structure/Communication/ST_MasterJointData.TcDUT
// Output from master arm control task 
// Input to safety task and force controller task
TYPE ST_MasterJointData :
STRUCT
	// joint position compute with motor encoder
	m_curMotorPos :ARRAY[1..g_mArmNum] OF Vec7d;
	
	// joint position compute with link/abs encoder
	m_curLinkPos :ARRAY[1..g_mArmNum] OF Vec7d;
	
	// target joint position 
	m_cmdJntPos :ARRAY[1..g_mArmNum] OF Vec7d;
	
	// current joint position 
	m_curJntPos :ARRAY[1..g_mArmNum] OF Vec7d;
	
	// target joint velocity 
	m_cmdJntVel :ARRAY[1..g_mArmNum] OF Vec7d;
	
	// current joint position 
	m_curJntVel :ARRAY[1..g_mArmNum] OF Vec7d;
	
	// command joint torque 
	m_cmdJntTrq :ARRAY[1..g_mArmNum] OF Vec7d;
	
	// current joint torque 
	m_curJntTrq :ARRAY[1..g_mArmNum] OF Vec7d;
	
END_STRUCT
END_TYPE

// ---- DUTs/Structure/Communication/ST_SlaveStatus.TcDUT
// Output from Controller
// Input to master arm control task
TYPE ST_SlaveStatus :
STRUCT
	
	// state machine
	m_armState:ARRAY[1..g_sArmNum] OF E_SlaveArmState:=[g_sArmNum(SlaveArmState_Init)];
	
	// instrument info
	m_instruStauts :ARRAY[1..g_sArmNum] OF ST_InstruStatus;
	
	// command arm pose in endoscope view
	m_cmdArmPose:ARRAY[1..g_sArmNum] OF ST_Frame;
	
	// current arm pose in endoscope view
	m_curArmPose:ARRAY[1..g_sArmNum] OF ST_Frame;
	
	// command arm twist[linear velocity; angular veloicty] in endoscope view
	m_cmdArmTwist:ARRAY[1..g_sArmNum] OF Vec6d;
	
	// current arm twist[linear velocity; angular veloicty] in endoscope view
	m_curArmTwist:ARRAY[1..g_sArmNum] OF vec6d;

END_STRUCT
END_TYPE

// ---- DUTs/Structure/Communication/ST_SlaveJointData.TcDUT
TYPE ST_SlaveJointData :
STRUCT
	
	// joint position compute with motor encoder
	m_curMotorPos :ARRAY[1..g_sArmNum, 1..g_sJntNum] OF LREAL;
	
	// joint position compute with link/abs encoder
	m_curLinkPos :ARRAY[1..g_sArmNum, 1..g_sJntNum] OF LREAL;
	
	// target joint position 
	m_cmdJntPos :ARRAY[1..g_sArmNum, 1..g_sJntNum] OF LREAL;
	
	// current joint position 
	m_curJntPos :ARRAY[1..g_sArmNum, 1..g_sJntNum] OF LREAL;
	
	// target joint velocity 
	m_cmdJntVel :ARRAY[1..g_sArmNum, 1..g_sJntNum] OF LREAL;
	
	// current joint position 
	m_curJntVel :ARRAY[1..g_sArmNum, 1..g_sJntNum] OF LREAL;
	
	// command joint torque 
	m_cmdJntTrq :ARRAY[1..g_sArmNum, 1..g_sJntNum] OF LREAL;
	
	// current joint torque 
	m_curJntTrq :ARRAY[1..g_sArmNum, 1..g_sJntNum] OF LREAL;
END_STRUCT
END_TYPE

// ---- DUTs/Structure/ST_ArmCtrlCmds.TcDUT
TYPE ST_ArmCtrlCmds :
STRUCT
	// arm control data
	m_jntEnableFlag : Vec7i;
	m_jntOPMode : Vec7i;
	m_cmdJntPos : VEC7d;
	m_cmdJntVel : VEC7d;
	m_cmdJntAcc : VEC7d;
	m_cmdJntTrq : VEC7d;
	m_cmdCartPose : ST_Frame;
	m_cmdCartTwist : Vec6d;
	
END_STRUCT
END_TYPE

// ---- DUTs/Structure/ST_MasterInputDataPool.TcDUT
// Struct contains all data from other tasks and controller used for master control
TYPE ST_MasterInputDataPool :
STRUCT
		
	// UI information, import from UI controller
	m_UIData AT %I*:ST_UIData;
	
	// safety information, import from safety check task
	m_safetyData AT %I*: ST_CartStatus;
	
	// cart information, import from other task
	m_cartStatus AT %I*:ST_CartStatus;
	
	// slave robot information, import from other device
	m_slaveStatus AT %I*:ST_SlaveStatus;
	
	// master dynamic data
	m_masterDynaData AT %I* : ST_MasterDynaData;
	
END_STRUCT
END_TYPE

// ---- DUTs/Type/Mat67.TcDUT
TYPE Mat67 : ARRAY[1..6, 1..7] OF LREAL; END_TYPE

// ---- DUTs/Type/Mat6d.TcDUT
TYPE Mat6d : ARRAY[1..6, 1..6] OF LREAL; END_TYPE

// ---- DUTs/Type/Mat76.TcDUT
TYPE Mat76 : ARRAY[1..7, 1..6] OF LREAL; END_TYPE

// ---- DUTs/Type/Mat7d.TcDUT
TYPE Mat7d : ARRAY[1..7, 1..7] OF LREAL; END_TYPE

// ---- DUTs/Enum/E_DriverStatusWord.TcDUT
TYPE E_DriverStatusWord :
(
	DriverStatusWord_INIT := 4641,
	DriverStatusWord_PREOP := 4659,
	DriverStatusWord_OP := 4663
);
END_TYPE

// ---- DUTs/Enum/E_SlaveArmState.TcDUT
TYPE E_SlaveArmState :
(
	SlaveArmState_Error := 1,
	SlaveArmState_Init :=2,
	SlaveArmState_Standby :=3,
	SlaveArmState_InstallPanel:=4,
	SlaveArmState_PanelReady :=5,
	SlaveArmState_InstallInstru :=6,
	SlaveArmState_InstruReady :=7,
	SlaveArmState_MasterSlave :=8,
	SlaveArmState_InstallScope :=9,
	SlaveArmState_ScopeReady :=10,
	SlaveArmState_EndoScope :=11,
	SlaveArmState_Cart := 12
);
END_TYPE

// ---- DUTs/Structure/ST_Frame.TcDUT
TYPE ST_Frame :
STRUCT
	m_pos :Vec3d :=g_zeroVec3d;
	m_rot :Mat3d :=g_eye3d;
END_STRUCT
END_TYPE

// ---- DUTs/Structure/ST_InstruStatus.TcDUT
TYPE ST_InstruStatus :
STRUCT
	
	m_ready:BOOL := FALSE;
	m_type : E_InstrumentType := InstruType_UNKNOWM;
	m_fingerAngle:LREAL := 0.0;
	
END_STRUCT
END_TYPE

// ---- DUTs/Type/Mat3d.TcDUT
TYPE Mat3d : ARRAY[1..3, 1..3] OF LREAL; END_TYPE

// ---- DUTs/Type/Vec3d.TcDUT
TYPE Vec3d : ARRAY[1..3] OF LREAL; END_TYPE

// ---- DUTs/Type/Vec6d.TcDUT
TYPE Vec6d : ARRAY[1..6] OF LREAL; END_TYPE

// ---- GVLs/GVL_ControlParameters.TcGVL
{attribute 'global_init_slot' := '49991'}
VAR_GLOBAL CONSTANT
	// master arm joint position controller parameters
	g_posKp :ARRAY[1..7] OF LREAL :=[0.0, 0.0, 0.0, 4.0, 0.0, 0.0, 0.0];
	g_posKd :ARRAY[1..7] OF LREAL :=[0.0, 0.0, 0.0, 0.1, 0.0, 0.0, 0.0];
	g_posKi :ARRAY[1..7] OF LREAL :=[0.0, 0.0, 0.0, 0.0, 0.0, 0.0, 0.0];
	g_posKiLimit :ARRAY[1..7] OF LREAL :=[500,500,500,500,100,100,100];// define in current
	g_posCtrlLimit :ARRAY[1..7] OF LREAL :=[1000,1000,1000,1000,200,200,200];// define in current
	
	// redundant joint4 following motion parameters
	g_jnt4MaxFollowVel :LREAL :=2*pi;
	g_jnt4MaxFollowAcc :LREAL :=6*pi;
	
	// control tolerance
	g_jntCtrlPosTol :LREAL :=0.2*g_deg2Rad;
	g_cartCtrlPosTol :LREAL :=0.0002;
	g_cartCtrlOriTol :LREAL :=0.2*g_deg2Rad;
	
	// filter cut-off frequency for velocity and torque
	g_curJntVelLpfCutoffFreq :LREAL := 30;
	g_cmdJntPosLpfCutoffFreq :LREAL := 30;
	g_cmdJntTrqLpfCutoffFreq :LREAL := 300;
	
	// controller would keep command unchanged when error 
	// between command and current value is less than this value
	g_jntCtrlErrForCmdHold :LREAL :=2.0*g_deg2Rad;
	
	// joint is assumed to be static if velocity is less than this value
	g_jntStaticVelThres :LREAL :=0.2*g_deg2Rad;
	
	// home motion parameters
	g_homePosture:ARRAY [1..2, 1..7] OF LREAL:=[0.0, -PI/2, 0, -PI, PI, -PI/2, 0,
							 			  			0.0, -PI/2, 0, 0, PI, PI/2, 0];
	g_homeMaxjntVel:Vec7d:=[1.0, 1.0, 1.0, 1.0, 1.0, 1.0, 1.0];
	g_homeMaxjntAcc:Vec7d:=[1.0, 1.0, 1.0, 2.0, 2.0, 2.0, 2.0];
	g_homeMaxjntJerk:Vec7d:=[7(4.0)];
END_VAR

// ---- GVLs/GVL_JointEncoderCaliData.TcGVL
VAR_GLOBAL CONSTANT
	// abolute encoder expanded limit buffer in case there is calibrtion error at limit position
	g_linkEncLimitBuffer : DINT := 5000;
	
	// absolute encoder value at minimal joint positon
	g_minLinkEncoder :ARRAY[1..g_mArmNum, 1..g_mJntNum] OF DINT :=
		[8989196, 4134520, 15344624, 1912720, 16331520, 14419696, 0,
		 13092100, 9431568, 8498692, 8222800, 659040, 8986672, 0];
		 
	// absolute encoder value at maximum joint positon
	g_maxLinkEncoder :ARRAY[1..g_mArmNum, 1..g_mJntNum] OF DINT :=
		[14678512, 15070764, 1808188, 7240592, 12225952, 1889888, 16777216,
		 2006608, 3571264, 12804156, 13448864, 13314448, 13295680, 16777216];
	
	// absolute encoder value at calibrated positon
	g_caliLinkEncoder :ARRAY[1..g_mArmNum, 1..g_mJntNum] OF DINT :=
		[11841020, 1344500, 110836, 11640160, 5911600, 16609560, 9605344,
		 15937870, 6515250, 10128280, 4044030, 7101400, 11107232, 8959776];
	
	 // if absolute encoder value cross zeros within joint motion range
	 // NOTICE: joint 7 is always 0.
	g_linkEncZeroCross :ARRAY[1..g_mArmNum, 1..g_mJntNum] OF INT :=
		[0, 1, 1, 1, 1, 1, 0,
		 1, 0, 1, 1, 0, 0, 0];
	
	// flag if joint can rotate multiple cycles
	g_multipleCyclesJoint :ARRAY[1..g_mArmNum, 1..g_mJntNum] OF INT :=
		[0, 0, 0, 0, 0, 0, 1,
		 0, 0, 0, 0, 0, 0, 1];
		 
	// joint position at link encoder calibrated point
	g_linkEncCaliJntPos :ARRAY[1..g_mArmNum, 1..g_mJntNum] OF LREAL :=
		[0.0, -PI/2, 0.0, -pi, pi, -PI/2, 0.0,
		 0.0, -PI/2, 0.0, 0.0, pi, PI/2, 0.0];
END_VAR

// ---- GVLs/GVL_MathDefine.TcGVL
VAR_GLOBAL CONSTANT
	g_smallNum :LREAL := 1E-6;
	g_largeNum: LREAL :=1E16;
	g_deg2Rad :LREAL := pi/180.0;
	g_rad2Deg :LREAL := 180.0/pi;
	
	g_eye3d :Mat3d:=[1, 0, 0,
					 0, 1, 0,
					 0, 0, 1];
	g_zeorMat3d :Mat3d:=[9(0)];
	
	g_zeroMat6d :Mat6d:=[36(0)];
	g_zeroMat7d :Mat7d:=[49(0)];
	g_eye7d :Mat7d:=[1, 0, 0, 0, 0, 0, 0, 
					 0, 1, 0, 0, 0, 0, 0, 
					 0, 0, 1, 0, 0, 0, 0, 
					 0, 0, 0, 1, 0, 0, 0,
					 0, 0, 0, 0, 1, 0, 0,
					 0, 0, 0, 0, 0, 1, 0,
					 0, 0, 0, 0, 0, 0, 1];
	
	g_zeroVec3d :Vec3d:= [3(0)];
	g_onesVec3d: Vec3d:=[3(1)];
	
	g_zeroVec6d: Vec6d:=[6(0)];
	g_onesVec6d: Vec6d:=[6(1)];
	
	g_zeroVec7d: Vec7d:=[7(0)];
	g_onesVec7d: Vec7d:=[7(1.0)];
	g_zeroVec7i: Vec7i:=[7(0)];
	g_onesVec7i: Vec7i:=[7(1)];
	
	g_allPosMode:Vec7i:=[7(DriverOPMode_Pos)];
	g_allTrqMode:Vec7i:=[7(DriverOPMode_Trq)];
	g_allPosTrqMode:Vec7i:=[7(DriverOPMode_PosTrq)];
	
	
END_VAR

// ---- GVLs/GVL_MotorParameters.TcGVL
{attribute 'global_init_slot' := '49991'}
VAR_GLOBAL CONSTANT
	// encoder resolution
	g_incEncoderRes :ARRAY[1..7] OF DINT :=[7(65536)];
	g_absEncoderRes :ARRAY[1..7] OF DINT :=[7(16777216)];
	
	// reduction ratio
	g_motorReduction :ARRAY[1..7] OF LREAL :=[43.9658,26.859,26.8018,(66.0/10)*3,4554.0/130, 4554.0/130,5625.0/361];
	g_absEncoderReduction :ARRAY[1..7] OF LREAL :=[7(1.0)];
	
	// motor parameters
	g_motorTrqConst :ARRAY[1..7] OF LREAL :=[0.0538,0.0538,0.0538,0.0299,0.0193,0.0193,0.0193];
	g_motorMaxCurrent :ARRAY[1..7] OF LREAL :=[1000,1000,1000,1010,204,204,204];//mA
	
	// motor and absEncoder direction
	g_motorDir :ARRAY[1..2, 1..7] OF INT :=[1, 1, -1, 1, 1, -1, -1,	
											1, 1, -1, 1, 1, -1, -1];
	g_asbEncoderDir :ARRAY[1..2, 1..7] OF INT :=[-1, -1, 1, -1, 1, 1, 1,
												 -1, -1, 1, -1, 1, 1, 1];
																 
	// joint position limit
	g_minJntPos: ARRAY[1..2,1..7] OF LREAL:=[-60*g_deg2Rad,	-45*g_deg2Rad-pi/2,		-45*g_deg2Rad, 	-2*pi, 	-135*g_deg2Rad+pi,		-45*g_deg2Rad-pi/2,		-340*g_deg2Rad,
											 								-60*g_deg2Rad,	-45*g_deg2Rad-pi/2,		-45*g_deg2Rad,	-pi,		-135*g_deg2Rad+pi,		-45*g_deg2Rad+pi/2,	-340*g_deg2Rad];
	g_maxJntPos: ARRAY[1..2,1..7] OF LREAL:=[60*g_deg2Rad,	60*g_deg2Rad-pi/2,		60*g_deg2Rad,		0,			135*g_deg2Rad+pi,		45*g_deg2Rad-pi/2,		340*g_deg2Rad,
								             								 60*g_deg2Rad,	60*g_deg2Rad-pi/2,		60*g_deg2Rad,		pi,			135*g_deg2Rad+pi,		45*g_deg2Rad+pi/2,		340*g_deg2Rad];
	
	// joint velocity limit
	g_maxJntVel :ARRAY[1..7] OF LREAL :=[7(2*pi)];
	
END_VAR

// ---- GVLs/GVL_SystemParameters.TcGVL
VAR_GLOBAL CONSTANT
	
	g_mArmNum :INT := 2;	
	g_mJntNum :INT := 7;	
	g_sArmNum :INT := 4;	
	g_sJntNum :INT := 11;
	g_cartDofs :INT :=6;
	
	
	
	// control loop interval for each task
	g_armControlLoopInterval :LREAL :=0.001;
	g_armControlFreq :LREAL :=1.0/g_armControlLoopInterval;
	g_armDynamicLoopInterval :LREAL := 0.001;
	g_armDynamicFreq :LREAL := 1.0/g_armDynamicLoopInterval;
	g_cartControlLoopInterval :LREAL := 0.001;
	g_cartControlFreq :LREAL := 1.0/g_cartControlLoopInterval;
	
	// wait time before robot init  for ethercat to stablize 
	g_robotInitWaitTime : LREAL := 1.0;

END_VAR

// ---- FBs_StateControllers/I_MasterArmCtrl.TcIO
INTERFACE I_MasterArmCtrl

PROPERTY isFinished : bool
GET
END_GET
END_PROPERTY

METHOD reset : BOOL
VAR_INPUT
END_VAR
END_METHOD

METHOD run : BOOL
VAR_INPUT
	monitorAngle :LREAL;
	slaveIdx :INT;
END_VAR

VAR_IN_OUT CONSTANT
	i_masterArm :FB_MasterArm;
	i_slaveStatus :ST_SlaveStatus;
END_VAR
VAR_IN_OUT
	r_masterArmCtrlCmd :ST_ArmCtrlCmds;
END_VAR
END_METHOD

END_INTERFACE

// ---- Mains/MasterArmControl.TcPOU
PROGRAM MasterArmControl
VAR
	// flag to init robot
	m_robotInit :BOOL :=FALSE;
	
	// wait time before robot init  for ethercat to be statble 
	m_robotInitWaitTime : LREAL:=0;
	
	// master robot
	m_masterRobot:FB_MasterRobot;
	
	// master robot information, including arm status and cartesian data
	m_masterStatus AT %Q* :ST_MasterStatus;
	
	// master robot joint data
	m_masterJointsData AT %Q* :ST_MasterJointData;
	
	// all data from other tasks and controller 
	m_masterInputDataPool : ST_MasterInputDataPool;
	
	// code execute time measure
	m_codeTime : Profiler;
END_VAR

m_codeTime(START:=TRUE, RESET:=TRUE);

// wait communication to be stable
IF(m_robotInitWaitTime<g_robotInitWaitTime) THEN
	m_robotInitWaitTime := m_robotInitWaitTime+g_armControlLoopInterval;
	RETURN;
END_IF

// robot init
IF m_robotInit =FALSE THEN
	m_masterRobot.Init();
	m_robotInit:=TRUE;
END_IF

// robot run
m_masterRobot.run(m_masterInputDataPool);

// update data pool
m_masterRobot.getStatus(m_masterStatus,m_masterJointsData);

m_codeTime(START:=FALSE);

END_PROGRAM

// ---- FBs_Robots/FB_MasterRobot.TcPOU
FUNCTION_BLOCK FB_MasterRobot
VAR_INPUT
END_VAR
VAR_OUTPUT
END_VAR
VAR
	// master-slave motion scale
	m_motionScale :LREAL;
	
	// monitor angle
	m_monitorAngle :LREAL;
	
	// master arms, responsible for arm kinematic and control
	m_masterArms :ARRAY[1..g_mArmNum] OF FB_MasterArm;
	
	// arm state
	m_masterArmState:ARRAY[1..g_mArmNum] OF E_masterArmState:=[E_masterArmState.MasterArmState_Init,E_masterArmState.MasterArmState_Init];
	m_lastMasterArmState:ARRAY[1..g_mArmNum] OF E_masterArmState:=[E_masterArmState.MasterArmState_Init,E_masterArmState.MasterArmState_Init];
	m_nextMasterArmState:ARRAY[1..g_mArmNum] OF E_masterArmState:=[E_masterArmState.MasterArmState_Init,E_masterArmState.MasterArmState_Init];
	
	// index(1 to 4) of slave arm which is tele-linked to master arm
	m_teleSlaveArmIdx:ARRAY[1..g_mArmNum] OF E_MatchedSlaveArmIdx:=[MatchedSlaveArmIdx_NULL, MatchedSlaveArmIdx_null];
	
	// all arm controller instance 
	m_armCtrlFactory :ARRAY[1..g_mArmNum,1..MasterArmState_totalNum] OF I_MasterArmCtrl;
	m_armError :ARRAY[1..g_mArmNum] OF FB_ArmError;
	m_armInit :ARRAY[1..g_mArmNum] OF FB_ArmInit;
	m_armHome :ARRAY[1..g_mArmNum] OF FB_ArmHome;
	m_armStandBy :ARRAY[1..g_mArmNum] OF FB_ArmStandBy;
	m_armMatching :ARRAY[1..g_mArmNum] OF FB_ArmMatching;
	m_armReady :ARRAY[1..g_mArmNum] OF FB_ArmReady;
	m_armMasterSlave :ARRAY[1..g_mArmNum] OF FB_ArmMasterSlave;
	m_armClutch :ARRAY[1..g_mArmNum] OF FB_ArmClutch;
	m_armEndoscope :ARRAY[1..g_mArmNum] OF FB_ArmEndoscope;
	m_armCart :ARRAY[1..g_mArmNum] OF FB_ArmCart;
	
	// arm controller interface
	m_armCtrl :ARRAY[1..g_mArmNum] OF I_MasterArmCtrl;
	m_armCtrlCmds :ARRAY[1..g_mArmNum] OF ST_ArmCtrlCmds;

END_VAR

METHOD PUBLIC getStatus : BOOL
VAR_IN_OUT
	// master robot information, including arm status and cartesian data
	r_masterStatus :ST_MasterStatus;
	
	// master robot joint data
	r_masterJointsData :ST_MasterJointData;
	
END_VAR

VAR
	i:INT;
END_VAR
r_masterStatus.m_motionScale := m_motionScale;
r_masterStatus.m_armState:=m_masterArmState;
r_masterStatus.m_teleSlaveArmIdx := m_teleSlaveArmIdx;

// TODO: project cartesion data to monitor coordinate
FOR i:=1 TO g_mArmNum DO
	// current info
	r_masterStatus.m_gripAngle[i]:=m_masterArms[i].gripAngle;
	// cartesion
	r_masterStatus.m_curArmPose[i]:=m_masterArms[i].curCartPose;
	r_masterStatus.m_curArmTwist[i]:=m_masterArms[i].curCartTwist;
	// joint
	r_masterJointsData.m_curMotorPos[i]:=m_masterArms[i].curMotorPos;
	r_masterJointsData.m_curLinkPos[i]:=m_masterArms[i].curLinkPos;
	r_masterJointsData.m_curJntPos[i]:=m_masterArms[i].curJntPos;
	r_masterJointsData.m_curJntVel[i]:=m_masterArms[i].curJntVel;
	r_masterJointsData.m_curJntTrq[i]:=m_masterArms[i].curJntTrq;
	
	// command info
	// cartesion
	r_masterStatus.m_cmdArmPose[i]:=m_armCtrlCmds[i].m_cmdCartPose;
	r_masterStatus.m_cmdArmTwist[i]:=m_armCtrlCmds[i].m_cmdCartTwist;
	// joint info
	r_masterJointsData.m_cmdJntPos[i]:=m_armCtrlCmds[i].m_cmdJntPos;
	r_masterJointsData.m_cmdJntVel[i]:=m_armCtrlCmds[i].m_cmdJntVel;
	r_masterJointsData.m_cmdJntTrq[i]:=m_armCtrlCmds[i].m_cmdJntTrq;
	
END_FOR
END_METHOD

METHOD PUBLIC Init : BOOL
VAR_INPUT
END_VAR
VAR
	i:INT;
END_VAR
FOR i:=1 TO g_mArmNum DO
	// arm init
	m_masterArms[i].Init(i);
	m_masterArmState[i]:=MasterArmState_Init;
	m_lastMasterArmState[i]:=MasterArmState_Init;
	m_nextMasterArmState[i]:=MasterArmState_Init;
	m_teleSlaveArmIdx[i]:=MatchedSlaveArmIdx_NULL;
	
	// command init
	m_armCtrlCmds[i].m_jntEnableFlag := g_zeroVec7i;
	m_armCtrlCmds[i].m_jntOPMode := g_allPosMode;
	m_armCtrlCmds[i].m_cmdCartPose := m_masterArms[i].curCartPose;
	m_armCtrlCmds[i].m_cmdCartTwist := g_zeroVec6d;
	m_armCtrlCmds[i].m_cmdJntPos := m_masterArms[i].curJntPos;
	m_armCtrlCmds[i].m_cmdJntVel := g_zeroVec7d;
	m_armCtrlCmds[i].m_cmdJntAcc := g_zeroVec7d;
	m_armCtrlCmds[i].m_cmdJntTrq := g_zeroVec7d;
	
	// generate controller factory
	m_armCtrlFactory[i,MasterArmState_Error] := m_armError[i];
	m_armCtrlFactory[i,MasterArmState_Init] := m_armInit[i];
	m_armCtrlFactory[i,MasterArmState_Home] := m_armHome[i];
	m_armCtrlFactory[i,MasterArmState_Standby] := m_armStandBy[i];
	m_armCtrlFactory[i,MasterArmState_Matching] := m_armMatching[i];
	m_armCtrlFactory[i,MasterArmState_Ready] := m_armReady[i];
	m_armCtrlFactory[i,MasterArmState_MasterSlave] := m_armMasterSlave[i];
	m_armCtrlFactory[i,MasterArmState_Clutch] := m_armClutch[i];
	m_armCtrlFactory[i,MasterArmState_Endoscope] := m_armEndoscope[i];
	m_armCtrlFactory[i,MasterArmState_Cart] := m_armCart[i];

	// assign controller
	m_armCtrl[i]:=m_armCtrlFactory[i,m_masterArmState[i]];
END_FOR
END_METHOD

METHOD PUBLIC run : BOOL
VAR_IN_OUT CONSTANT
	i_masterInputDataPool:ST_MasterInputDataPool;
END_VAR
VAR
	i:INT;
END_VAR
m_motionScale := i_masterInputDataPool.m_UIData.m_motionScale;
m_monitorAngle := i_masterInputDataPool.m_cartStatus.m_monitorAngle;

// state machine transition
stateMachine(i_masterInputDataPool);

FOR i:=1 TO g_mArmNum DO
	// update dynamic data
	m_masterArms[i].updateDyna(i_masterInputDataPool.m_masterDynaData);
								
	// update master arm kinematics
	m_masterArms[i].updateStatus();
	
	// null ptr check
	IF 0 = m_armCtrl[i] THEN
		EXIT;
	END_IF
	
	// run controller
	m_armCtrl[i].run(m_monitorAngle, m_teleSlaveArmIdx[i], m_masterArms[i],
						i_masterInputDataPool.m_slaveStatus,m_armCtrlCmds[i]);

	// update commands to drivers
	m_masterArms[i].updateCmds(m_armCtrlCmds[i]);

END_FOR
END_METHOD

// state machine check and transit 
METHOD PROTECTED stateMachine : BOOL
VAR_IN_OUT CONSTANT
		i_masterInputDataPool:ST_MasterInputDataPool;
END_VAR
VAR
	i:INT;
END_VAR
FOR i:=1 TO g_mArmNum DO
	// State machine transit 
	CASE m_masterArmState[i] OF
		// init
		MasterArmState_Init:
			IF m_armCtrl[i].isFinished  THEN
				// NOTICE: multiple cycles joints back to center during initialization
				// 			need to reset joints encoder data again
				m_masterArms[i].initJntPos();
				
				m_nextMasterArmState[i]:=MasterArmState_Home;
			END_IF

		//home
		MasterArmState_Home:
			IF m_armCtrl[i].isFinished  THEN
				m_nextMasterArmState[i]:=MasterArmState_Standby;
			END_IF
		
		//standby
(*		MasterArmState_Standby:
		
		//matching
		MasterArmState_Matching:
		
		//ready
		MasterArmState_Ready:
		
		//MasterSlave
		MasterArmState_MasterSlave:*)
	END_CASE
	
	// Controller transit
	IF m_nextMasterArmState[i]<> m_masterArmState[i] THEN
		// reset current controller
		m_armCtrl[i].reset();
		
		// transit to new one
		m_lastMasterArmState[i]:=m_masterArmState[i];
		m_masterArmState[i]:=m_nextMasterArmState[i];
		m_armCtrl[i]:=m_armCtrlFactory[i,m_masterArmState[i]];
	END_IF
END_FOR
END_METHOD

END_FUNCTION_BLOCK

// ---- FBs_Robots/FB_MasterArm.TcPOU
FUNCTION_BLOCK FB_MasterArm
// NOTICE: all joints are the ture active joints, not DH ones!
VAR_INPUT
END_VAR
VAR_OUTPUT
END_VAR
VAR
	// arm index, 0 for left arm, 1 for right arm
	m_armIdx: INT;
	
	// grip angle from hall sensor IO
	m_gripHallSensorValue AT%I* :UDINT;
	m_gripAngle :LREAL;
	
	// arm block
	m_joints :ARRAY[1..g_mJntNum] OF FB_Joint;
	
	// arm cartesian data, defined in each arm origin
	m_curCartPose	:ST_Frame;
	m_curCartTwist: Vec6d;
	
	// arm joint data
	m_curMotorPos :Vec7d;
	m_curLinkPos :Vec7d;
	m_curJntPos :Vec7d;
	m_curJntVel :Vec7d;
	m_curJntTrq :Vec7d;
	m_jntCtrlTrq :Vec7d;
	
	// arm daynamic data
	m_jntGravity : Vec7d;
	m_jntMassMat : Mat7d;
	m_lambda :Mat6d;
	m_dynaNullspace :Mat7d;
	
	// arm jacobian 
	m_jaco :ARRAY[1..g_cartDofs, 1..g_mJntNum] OF LREAL;
	
	// joint position controller
	m_jntPIDCtrl :ARRAY[1..g_mJntNum] OF FB_PID;
	
END_VAR

PROPERTY armIdx : int
GET
armIdx:=m_armIdx;
END_GET
END_PROPERTY

// TODO
METHOD PROTECTED calcGripAngle : LREAL
VAR_INPUT
END_VAR
END_METHOD

METHOD PUBLIC calcJaco : BOOL
VAR_IN_OUT CONSTANT
	i_jntPos :ARRAY[1..g_mJntNum] OF LREAL;
END_VAR
VAR_IN_OUT
	r_jaco :ARRAY[1..g_cartDofs, 1..g_mJntNum] OF LREAL;
END_VAR
VAR_INPUT
END_VAR

VAR
	q1,q2, q3, q4, q5, q6, q7 :LREAL;
	d1,d4,a3,a4 :LREAL;
	j:INT;
END_VAR
// !Convert active joint position to DH model for kinematic calculation
q1:=i_jntPos[1];  
q2:=i_jntPos[2];  
q3:=i_jntPos[3]-i_jntPos[2];  //q3=q8-q2
q4:=i_jntPos[4]+i_jntPos[3]-i_jntPos[2]-pi/2;//q4DH=q4motor+q8-q2-90;  
q5:=i_jntPos[5];  
q6:=i_jntPos[6];  
q7:=i_jntPos[7];  
d1:=g_d1;
d4:=g_d4;
a3:=g_a3;
a4:=g_a4;

// jacobian with DH joints
r_jaco[1,1]:=-SIN(q1)*(COS(q2)*(a3 + a4*COS(q3) - d4*SIN(q3)) - SIN(q2)*(d4*COS(q3) + a4*SIN(q3))) ;
r_jaco[1,2]:=-COS(q1)*(SIN(q2)*(a3 + a4*COS(q3) - d4*SIN(q3)) + COS(q2)*(d4*COS(q3) + a4*SIN(q3))) ;
r_jaco[1,3]:=-COS(q1)*(d4*COS(q2 + q3) + a4*SIN(q2 + q3)) ;
r_jaco[1,4]:=0 ;
r_jaco[1,5]:=0 ;
r_jaco[1,6]:=0 ;
r_jaco[1,7]:=0;
 
r_jaco[2,1]:=COS(q1)*(COS(q2)*(a3 + a4*COS(q3) - d4*SIN(q3)) - SIN(q2)*(d4*COS(q3) + a4*SIN(q3))); 
r_jaco[2,2]:=-SIN(q1)*(SIN(q2)*(a3 + a4*COS(q3) - d4*SIN(q3)) + COS(q2)*(d4*COS(q3) + a4*SIN(q3))); 
r_jaco[2,3]:=-SIN(q1)*(d4*COS(q2 + q3) + a4*SIN(q2 + q3)); 
r_jaco[2,4]:=0; 
r_jaco[2,5]:=0; 
r_jaco[2,6]:=0; 
r_jaco[2,7]:=0;

 
r_jaco[3,1]:=0 ;
r_jaco[3,2]:=- COS(q1)*(COS(q1)*COS(q2)*(a3 + a4*COS(q3) - d4*SIN(q3)) - COS(q1)*SIN(q2)*(d4*COS(q3) + a4*SIN(q3))) - SIN(q1)*(COS(q2)*SIN(q1)*(a3 + a4*COS(q3) - d4*SIN(q3)) - SIN(q1)*SIN(q2)*(d4*COS(q3) + a4*SIN(q3)));
r_jaco[3,3]:=- COS(q1)*(a4*COS(q2 + q3)*COS(q1) - d4*SIN(q2 + q3)*COS(q1)) - SIN(q1)*(a4*COS(q2 + q3)*SIN(q1) - d4*SIN(q2 + q3)*SIN(q1));
r_jaco[3,4]:=0;
r_jaco[3,5]:=0;
r_jaco[3,6]:=0 ;
r_jaco[3,7]:=0 ;

r_jaco[4,1]:=0 ;
r_jaco[4,2]:=-SIN(q1) ;
r_jaco[4,3]:=-SIN(q1) ;
r_jaco[4,4]:=-SIN(q2 + q3)*COS(q1) ;
r_jaco[4,5]:=COS(q2 + q3)*COS(q1)*SIN(q4) - COS(q4)*SIN(q1) ;
r_jaco[4,6]:=- SIN(q5)*(SIN(q1)*SIN(q4) + COS(q2 + q3)*COS(q1)*COS(q4)) - SIN(q2 + q3)*COS(q1)*COS(q5) ;
r_jaco[4,7]:=SIN(q6)*(COS(q5)*(SIN(q1)*SIN(q4) + COS(q4)*(COS(q1)*COS(q2)*COS(q3) - COS(q1)*SIN(q2)*SIN(q3))) - SIN(q5)*(COS(q1)*COS(q2)*SIN(q3) + COS(q1)*COS(q3)*SIN(q2))) - COS(q6)*(COS(q4)*SIN(q1) - SIN(q4)*(COS(q1)*COS(q2)*COS(q3) - COS(q1)*SIN(q2)*SIN(q3)));
 
r_jaco[5,1]:=0; 
r_jaco[5,2]:=COS(q1); 
r_jaco[5,3]:=COS(q1); 
r_jaco[5,4]:=-SIN(q2 + q3)*SIN(q1); 
r_jaco[5,5]:=COS(q1)*COS(q4) + COS(q2 + q3)*SIN(q1)*SIN(q4); 
r_jaco[5,6]:=SIN(q5)*(COS(q1)*SIN(q4) - COS(q2 + q3)*COS(q4)*SIN(q1)) - SIN(q2 + q3)*COS(q5)*SIN(q1); 
r_jaco[5,7]:=COS(q6)*(COS(q1)*COS(q4) - SIN(q4)*(SIN(q1)*SIN(q2)*SIN(q3) - COS(q2)*COS(q3)*SIN(q1))) - SIN(q6)*(COS(q5)*(COS(q1)*SIN(q4) + COS(q4)*(SIN(q1)*SIN(q2)*SIN(q3) - COS(q2)*COS(q3)*SIN(q1))) + SIN(q5)*(COS(q2)*SIN(q1)*SIN(q3) + COS(q3)*SIN(q1)*SIN(q2)));

r_jaco[6,1]:=1 ;
r_jaco[6,2]:=0 ;
r_jaco[6,3]:=0 ;
r_jaco[6,4]:=-COS(q2 + q3) ;
r_jaco[6,5]:=-SIN(q2 + q3)*SIN(q4) ;
r_jaco[6,6]:=SIN(q2 + q3)*COS(q4)*SIN(q5) - COS(q2 + q3)*COS(q5) ;
r_jaco[6,7]:=- SIN(q6)*(COS(q2 + q3)*SIN(q5) + SIN(q2 + q3)*COS(q4)*COS(q5)) - SIN(q2 + q3)*COS(q6)*SIN(q4);

// jacobian with active joints
// jaco_DH*qdot_DH = jaco_DH * (A * qdot)= jaco * qdot
// A =[ 1  0 0 0 0 0 0
//		0  1 0 0 0 0 0
//		0 -1 1 0 0 0 0
//		0 -1 1 1 0 0 0
//		0 0  0 0 1 0 0
//      0 0  0 0 0 1 0
// 		0 0  0 0 0 0 1]
 FOR j:=1 TO 6 DO 
	 r_jaco[j,2]:=r_jaco[j,2]-r_jaco[j,3]-r_jaco[j,4];
	 r_jaco[j,3]:=r_jaco[j,3]+r_jaco[j,4];
 END_FOR
END_METHOD

PROPERTY curCartPose : ST_Frame
GET
curCartPose :=m_curCartPose;
END_GET
END_PROPERTY

PROPERTY curCartTwist : Vec6d
GET
curCartTwist :=m_curCartTwist;
END_GET
END_PROPERTY

PROPERTY curJntPos : Vec7d
GET
curJntPos:=m_curJntPos;
END_GET
END_PROPERTY

PROPERTY curJntTrq : Vec7d
GET
curJntTrq:=m_curJntTrq;
END_GET
END_PROPERTY

PROPERTY curJntVel : Vec7d
GET
curJntVel:=m_curJntVel;
END_GET
END_PROPERTY

PROPERTY curLinkPos : Vec7d
GET
curLinkPos:=m_curLinkPos;
END_GET
END_PROPERTY

PROPERTY curMotorPos : Vec7d
GET
curMotorPos:=m_curMotorPos;
END_GET
END_PROPERTY

PROPERTY PUBLIC dynaNullspace : Mat7d
GET
dynaNullspace := m_dynaNullspace;
END_GET
END_PROPERTY

METHOD PUBLIC enable : BOOL
VAR_IN_OUT CONSTANT
	i_jntIdx :Vec7i;
END_VAR
VAR
	i :INT ;
END_VAR
FOR i:=1 TO g_mJntNum DO
	IF 1= i_jntIdx[i] THEN
		m_joints[i].enable();
	ELSE
		m_joints[i].disable();
	END_IF
END_FOR
END_METHOD

// from active joint position to cartesian pose in arm origin
METHOD PROTECTED forwardKinematic : BOOL
VAR_IN_OUT CONSTANT
	i_jntPos :ARRAY[1..g_mJntNum] OF LREAL;
END_VAR
VAR_IN_OUT
	r_curCartPose :ST_Frame;
END_VAR
VAR
	q1,q2, q3, q4, q5, q6, q7 :LREAL;
	d1,d4,a3,a4 :LREAL;
END_VAR
// !Convert active joint position to DH model for kinematic calculation
q1:=i_jntPos[1];  
q2:=i_jntPos[2];  
q3:=i_jntPos[3]-i_jntPos[2];  //q3=q8-q2
q4:=i_jntPos[4]+i_jntPos[3]-i_jntPos[2]-pi/2;//q4DH=q4motor+q8-q2-90;  
q5:=i_jntPos[5];  
q6:=i_jntPos[6];  
q7:=i_jntPos[7];  
d1:=g_d1;
d4:=g_d4;
a3:=g_a3;
a4:=g_a4;

// cartesian pose frame
r_curCartPose.m_pos[1]:=COS(q1)*(a4*COS(q2 + q3) - d4*SIN(q2 + q3) + a3*COS(q2)); 
r_curCartPose.m_pos[2]:=SIN(q1)*(a4*COS(q2 + q3) - d4*SIN(q2 + q3) + a3*COS(q2)); 
r_curCartPose.m_pos[3]:=d1 - d4*COS(q2 + q3) - a4*SIN(q2 + q3) - a3*SIN(q2); 
r_curCartPose.m_rot[1,1]:=COS(q7)*(SIN(q6)*(COS(q4)*SIN(q1) - SIN(q4)*(COS(q1)*COS(q2)*COS(q3) - COS(q1)*SIN(q2)*SIN(q3))) + COS(q6)*(COS(q5)*(SIN(q1)*SIN(q4) + COS(q4)*(COS(q1)*COS(q2)*COS(q3) - COS(q1)*SIN(q2)*SIN(q3))) - SIN(q5)*(COS(q1)*COS(q2)*SIN(q3) + COS(q1)*COS(q3)*SIN(q2)))) - SIN(q7)*(SIN(q5)*(SIN(q1)*SIN(q4) + COS(q4)*(COS(q1)*COS(q2)*COS(q3) - COS(q1)*SIN(q2)*SIN(q3))) + COS(q5)*(COS(q1)*COS(q2)*SIN(q3) + COS(q1)*COS(q3)*SIN(q2)));
r_curCartPose.m_rot[2,1]:=SIN(q7)*(SIN(q5)*(COS(q1)*SIN(q4) + COS(q4)*(SIN(q1)*SIN(q2)*SIN(q3) - COS(q2)*COS(q3)*SIN(q1))) - COS(q5)*(COS(q2)*SIN(q1)*SIN(q3) + COS(q3)*SIN(q1)*SIN(q2))) - COS(q7)*(SIN(q6)*(COS(q1)*COS(q4) - SIN(q4)*(SIN(q1)*SIN(q2)*SIN(q3) - COS(q2)*COS(q3)*SIN(q1))) + COS(q6)*(COS(q5)*(COS(q1)*SIN(q4) + COS(q4)*(SIN(q1)*SIN(q2)*SIN(q3) - COS(q2)*COS(q3)*SIN(q1))) + SIN(q5)*(COS(q2)*SIN(q1)*SIN(q3) + COS(q3)*SIN(q1)*SIN(q2))));
r_curCartPose.m_rot[3,1]:=- SIN(q7)*(COS(q2 + q3)*COS(q5) - SIN(q2 + q3)*COS(q4)*SIN(q5)) - COS(q7)*(COS(q2 + q3)*COS(q6)*SIN(q5) - SIN(q2 + q3)*SIN(q4)*SIN(q6) + SIN(q2 + q3)*COS(q4)*COS(q5)*COS(q6)); 
r_curCartPose.m_rot[1,2]:=- SIN(q7)*(SIN(q6)*(COS(q4)*SIN(q1) - SIN(q4)*(COS(q1)*COS(q2)*COS(q3) - COS(q1)*SIN(q2)*SIN(q3))) + COS(q6)*(COS(q5)*(SIN(q1)*SIN(q4) + COS(q4)*(COS(q1)*COS(q2)*COS(q3) - COS(q1)*SIN(q2)*SIN(q3))) - SIN(q5)*(COS(q1)*COS(q2)*SIN(q3) + COS(q1)*COS(q3)*SIN(q2)))) - COS(q7)*(SIN(q5)*(SIN(q1)*SIN(q4) + COS(q4)*(COS(q1)*COS(q2)*COS(q3) - COS(q1)*SIN(q2)*SIN(q3))) + COS(q5)*(COS(q1)*COS(q2)*SIN(q3) + COS(q1)*COS(q3)*SIN(q2))); 
r_curCartPose.m_rot[2,2]:=SIN(q7)*(SIN(q6)*(COS(q1)*COS(q4) - SIN(q4)*(SIN(q1)*SIN(q2)*SIN(q3) - COS(q2)*COS(q3)*SIN(q1))) + COS(q6)*(COS(q5)*(COS(q1)*SIN(q4) + COS(q4)*(SIN(q1)*SIN(q2)*SIN(q3) - COS(q2)*COS(q3)*SIN(q1))) + SIN(q5)*(COS(q2)*SIN(q1)*SIN(q3) + COS(q3)*SIN(q1)*SIN(q2)))) + COS(q7)*(SIN(q5)*(COS(q1)*SIN(q4) + COS(q4)*(SIN(q1)*SIN(q2)*SIN(q3) - COS(q2)*COS(q3)*SIN(q1))) - COS(q5)*(COS(q2)*SIN(q1)*SIN(q3) + COS(q3)*SIN(q1)*SIN(q2))); 
r_curCartPose.m_rot[3,2]:=SIN(q7)*(COS(q2 + q3)*COS(q6)*SIN(q5) - SIN(q2 + q3)*SIN(q4)*SIN(q6) + SIN(q2 + q3)*COS(q4)*COS(q5)*COS(q6)) - COS(q7)*(COS(q2 + q3)*COS(q5) - SIN(q2 + q3)*COS(q4)*SIN(q5)); 
r_curCartPose.m_rot[1,3]:=SIN(q6)*(COS(q5)*(SIN(q1)*SIN(q4) + COS(q4)*(COS(q1)*COS(q2)*COS(q3) - COS(q1)*SIN(q2)*SIN(q3))) - SIN(q5)*(COS(q1)*COS(q2)*SIN(q3) + COS(q1)*COS(q3)*SIN(q2))) - COS(q6)*(COS(q4)*SIN(q1) - SIN(q4)*(COS(q1)*COS(q2)*COS(q3) - COS(q1)*SIN(q2)*SIN(q3))); 
r_curCartPose.m_rot[2,3]:=COS(q6)*(COS(q1)*COS(q4) - SIN(q4)*(SIN(q1)*SIN(q2)*SIN(q3) - COS(q2)*COS(q3)*SIN(q1))) - SIN(q6)*(COS(q5)*(COS(q1)*SIN(q4) + COS(q4)*(SIN(q1)*SIN(q2)*SIN(q3) - COS(q2)*COS(q3)*SIN(q1))) + SIN(q5)*(COS(q2)*SIN(q1)*SIN(q3) + COS(q3)*SIN(q1)*SIN(q2)));
r_curCartPose.m_rot[3,3]:=- SIN(q6)*(COS(q2 + q3)*SIN(q5) + SIN(q2 + q3)*COS(q4)*COS(q5)) - SIN(q2 + q3)*COS(q6)*SIN(q4);
END_METHOD

PROPERTY gripAngle : LREAL
GET
gripAngle:=m_gripAngle;
END_GET
END_PROPERTY

METHOD PUBLIC init : BOOL
VAR_INPUT
	i_armIdx:INT;
END_VAR
VAR 
	i :INT ;
	currentRatioMotor2Jnt: LREAL;
END_VAR
// arm statues init
m_armIdx:=i_armIdx;
m_gripAngle:=0;

// joint init
FOR i:=1 TO g_mJntNum DO
	m_joints[i].init(m_armIdx, i);
END_FOR

// init joint encoder and position calculation
initJntPos();

// joint controller init
FOR i:=1 TO g_mJntNum DO 
	currentRatioMotor2Jnt:=g_motorTrqConst[i]*g_motorReduction[i]/1000;
	m_jntPIDCtrl[i].init(g_armControlLoopInterval,g_posKp[i],g_posKd[i],g_posKi[i],
		g_posKiLimit[i]* currentRatioMotor2Jnt,	g_posCtrlLimit[i]*currentRatioMotor2Jnt);
END_FOR

// compute current status
updateStatus();
END_METHOD

METHOD initJntPos : BOOL
VAR_INPUT
END_VAR
VAR
	i:INT ;
END_VAR
// joint init
FOR i:=1 TO g_mJntNum DO
	m_joints[i].initJntPos();
END_FOR

// link position of joint4 is influenced by joint2 and joint3, need to handle seperately
//q4DH=q4motor+q8-q2-90;  
m_joints[4].initLinkPos:= m_joints[4].initLinkPos-m_joints[3].initLinkPos+m_joints[2].initLinkPos+PI/2;
END_METHOD

// from cartesian pose in arm origin to active joint position
METHOD PUBLIC inverseKinematic : BOOL
VAR_INPUT
	q4:LREAL;
	solution_ID:INT;
END_VAR
VAR_IN_OUT CONSTANT
	i_curCartPose :ST_Frame;
END_VAR
VAR_IN_OUT
	r_jntPos :ARRAY[1..g_mJntNum] OF LREAL;
END_VAR
VAR
	a3,a4,d1,d4:LREAL;
	px,py,pz:lreal;
	nx,ny,nz:lreal;
	ox,oy,oz:lreal;
	ax,ay,az:lreal;

	q1,q2,q3,q5,q6,q7:LREAL;
	
	q11,q12:LREAL;
	k1,A,B,C,fi,R0,q21,q22:lreal;
	ins1,ins2:lreal;
	
	A11,A12,A21,A22,C1,C2:lreal;
	SIN23,COS23,q23:lreal;
	
	T_74_left_23,q61,q62:lreal;
	T_74_left_13,T_74_left_33:lreal;
	T_74_left_21,T_74_left_22:LREAL;	
	
	succeed_1,succeed_2,succeed:BOOL;
END_VAR


//***********************单臂逆向运动学**************************//
d1:=g_d1;
d4:=g_d4;
a3:=g_a3;
a4:=g_a4;

nx:=i_curCartPose.m_rot[1,1];  ny:=i_curCartPose.m_rot[2,1];  nz:=i_curCartPose.m_rot[3,1];
ox:=i_curCartPose.m_rot[1,2]; oy:=i_curCartPose.m_rot[2,2];  oz:=i_curCartPose.m_rot[3,2];
ax:=i_curCartPose.m_rot[1,3];  ay:=i_curCartPose.m_rot[2,3];  az:=i_curCartPose.m_rot[3,3];
px:=i_curCartPose.m_pos[1]; py:=i_curCartPose.m_pos[2]; pz:=i_curCartPose.m_pos[3];


//求解q1
q11:=atan2(y:= py, x:= px);
q12:=-q11;
IF (Solution_ID<=4) THEN
	q1:=q11;
ELSE
	q1:=q12;
END_IF



//求解q2
k1:=px*COS(q1) + py*SIN(q1);
A:=2*a3*pz - 2*a3*d1;
B:=2*a3*k1;
C:=a3*a3 - a4*a4 + d1*d1 - 2*d1*pz - d4*d4 + k1*k1 + pz*pz;
fi:=atan2(y:= B, x:= A);

R0:=SQRT(A*A+B*B);

//*************程序保护性处理，避免软件崩溃***************//
IF ABS(C/R0)>1 THEN
	succeed_1:=FALSE;
	succeed:=FALSE;
	RETURN;
ELSE
	succeed_1:=TRUE;
END_IF

ins1:=atan2(y:= C/R0, x:= SQRT(1-(C/R0)*(C/R0)));
q21:=fi-ins1;
ins2:=atan2(y:= C/R0, x:= -SQRT(1-(C/R0)*(C/R0)));
q22:=fi-ins2;

IF (Solution_ID=1) OR (Solution_ID=2) OR (Solution_ID=5) OR (Solution_ID=6) THEN
	q2:=q21;
ELSE
	q2:=q22;
END_IF




//求解q3
A11:=- d4;
A12:=a4;
A21:=- a4;
A22:=-d4;
C1:=k1- a3*COS(q2);
C2:=pz - d1 + a3*SIN(q2);
sin23:=(C1*A22-C2*A12)/(A11*A22-A21*A12);
cos23:=(C2*A11-C1*A21)/(A11*A22-A21*A12);
q23:=atan2(y:= sin23, x:= cos23);
q3:=q23-q2;




//求解q6
T_74_left_23:=ax*(COS(q4)*SIN(q1) - COS(q1)*COS(q2)*COS(q3)*SIN(q4) + COS(q1)*SIN(q2)*SIN(q3)*SIN(q4)) - ay*(COS(q1)*COS(q4) + COS(q2)*COS(q3)*SIN(q1)*SIN(q4) - SIN(q1)*SIN(q2)*SIN(q3)*SIN(q4)) + az*SIN(q2 + q3)*SIN(q4);

//*************程序保护性处理，避免软件崩溃***************//
IF ABS(T_74_left_23>1) THEN
	succeed_2:=FALSE;
	succeed:=FALSE;
	RETURN;
ELSE
	succeed_2:=TRUE;
END_IF

q61:=ACOS(-T_74_left_23);
q62:=-ACOS(-T_74_left_23);
IF (Solution_ID=1) OR (Solution_ID=3) OR (Solution_ID=5) OR (Solution_ID=7) THEN
	q6:=q61;
ELSE
	q6:=q62;
END_IF


//求解q5
T_74_left_13:=ax*(SIN(q1)*SIN(q4) + COS(q1)*COS(q2)*COS(q3)*COS(q4) - COS(q1)*COS(q4)*SIN(q2)*SIN(q3)) - ay*(COS(q1)*SIN(q4) - COS(q2)*COS(q3)*COS(q4)*SIN(q1) + COS(q4)*SIN(q1)*SIN(q2)*SIN(q3)) - az*SIN(q2 + q3)*COS(q4);
T_74_left_33:=- az*COS(q2 + q3) - ax*SIN(q2 + q3)*COS(q1) - ay*SIN(q2 + q3)*SIN(q1);
q5:=atan2(y:= T_74_left_33*SIN(q6), x:= T_74_left_13*SIN(q6));


//求解q7
T_74_left_21:=nx*(COS(q4)*SIN(q1) - COS(q1)*COS(q2)*COS(q3)*SIN(q4) + COS(q1)*SIN(q2)*SIN(q3)*SIN(q4)) - ny*(COS(q1)*COS(q4) + COS(q2)*COS(q3)*SIN(q1)*SIN(q4) - SIN(q1)*SIN(q2)*SIN(q3)*SIN(q4)) + nz*SIN(q2 + q3)*SIN(q4);
T_74_left_22:=ox*(COS(q4)*SIN(q1) - COS(q1)*COS(q2)*COS(q3)*SIN(q4) + COS(q1)*SIN(q2)*SIN(q3)*SIN(q4)) - oy*(COS(q1)*COS(q4) + COS(q2)*COS(q3)*SIN(q1)*SIN(q4) - SIN(q1)*SIN(q2)*SIN(q3)*SIN(q4)) + oz*SIN(q2 + q3)*SIN(q4);
q7:=atan2(y:= -T_74_left_22*SIN(q6), x:= T_74_left_21*SIN(q6));


//! convert DH joint postion to active joint position
r_jntPos[1]:=q1;
r_jntPos[2]:=q2;
r_jntPos[3]:=q3+q2; // q8 = q3+q2
r_jntPos[4]:=q4+q2-r_jntPos[3]+pi/2;//q4DH=q4motor+q8-q2-90;  
r_jntPos[5]:=q5;
r_jntPos[6]:=q6;
r_jntPos[7]:=q7;

succeed:=TRUE;
inverseKinematic:=succeed;
END_METHOD

METHOD PUBLIC isEnabled : BOOL
VAR_IN_OUT CONSTANT
	i_jntIdx :Vec7i;
END_VAR
VAR
	i :INT ;
END_VAR
isEnabled := TRUE;
FOR i:=1 TO g_mJntNum DO
	IF 1= i_jntIdx[i] THEN
		isEnabled :=  (m_joints[i].isEnabled() AND isEnabled);
	END_IF
END_FOR
END_METHOD

PROPERTY jntGravity : Vec7d
GET
jntGravity:=m_jntGravity;
END_GET
END_PROPERTY

PROPERTY PUBLIC massMat : Mat7d
GET
massMat :=m_jntMassMat;
END_GET
END_PROPERTY

// update joints control command
METHOD PUBLIC updateCmds : BOOL
VAR_IN_OUT CONSTANT
	i_armCtrlCmd : ST_ArmCtrlCmds;
END_VAR
VAR
	i:INT;
END_VAR
m_jntCtrlTrq:=i_armCtrlCmd.m_cmdJntTrq;

// enable/disable joints
enable(i_armCtrlCmd.m_jntEnableFlag);

// position/torque control
FOR i:=1 TO g_mJntNum DO 
	IF i_armCtrlCmd.m_jntOPMode[i]=DriverOPMode_PosTrq THEN
		// position controller and gravity feedforward
		m_jntCtrlTrq[i]:=m_jntPIDCtrl[i].run(i_armCtrlCmd.m_cmdJntPos[i],m_curJntPos[i],i_armCtrlCmd.m_cmdJntVel[i],m_curJntVel[i]);
		m_jntCtrlTrq[i]:=m_jntCtrlTrq[i]+m_jntGravity[i];
		m_joints[i].updateCmds(DriverOPMode_Trq,i_armCtrlCmd.m_cmdJntPos[i],m_jntCtrlTrq[i]);
	ELSIF i_armCtrlCmd.m_jntOPMode[i]=DriverOPMode_Trq THEN
		// gravity feedforward
		m_jntCtrlTrq[i]:=m_jntCtrlTrq[i]+m_jntGravity[i];
		m_joints[i].updateCmds(DriverOPMode_Trq,i_armCtrlCmd.m_cmdJntPos[i],m_jntCtrlTrq[i]);
	ELSE
		m_jntPIDCtrl[i].reset();
		m_jntCtrlTrq[i]:=0;
		m_joints[i].updateCmds(DriverOPMode_Pos,i_armCtrlCmd.m_cmdJntPos[i],m_jntCtrlTrq[i]);
	END_IF
	
END_FOR
END_METHOD

METHOD PUBLIC updateDyna : BOOL
VAR_IN_out constant
	masterDynaData : ST_MasterDynaData;
END_VAR
m_jntMassMat:=masterDynaData.m_massMat[m_armIdx];
m_lambda:=masterDynaData.m_lambda[m_armIdx];
m_dynaNullspace:=masterDynaData.m_dynaNullspace[m_armIdx];
m_jntGravity:=masterDynaData.m_gravity[m_armIdx];
END_METHOD

// update arm status, including kinematic and dynamic
METHOD PUBLIC updateStatus : BOOL
VAR_INPUT
END_VAR
VAR 
	i,j:INT;
END_VAR
// grip angle
m_gripAngle :=calcGripAngle();

// update joint data
FOR i:=1 TO g_mJntNum DO
	m_joints[i].updateStatus();
END_FOR

// get joint data
FOR i:=1 TO g_mJntNum DO
	m_curMotorPos[i]:=m_joints[i].motorPos;
	m_curLinkPos[i]:=m_joints[i].linkPos;
	m_curJntPos[i]:=m_joints[i].jntPos;
	m_curJntVel[i]:=m_joints[i].jntVel;
	m_curJntTrq[i]:=m_joints[i].jntTrq;
END_FOR 
//q4DH=q4motor+q8-q2-90;  
m_curLinkPos[4]:=m_curLinkPos[4]-m_curLinkPos[3]+m_curLinkPos[2]+PI/2;

// cartesion pose
forwardKinematic(m_curJntPos,m_curCartPose);

// jacobian
calcJaco(m_curJntPos,m_jaco);

// cartesian twist
m_curCartTwist:=Mat67Vec7(m_jaco,m_curJntVel);
END_METHOD

END_FUNCTION_BLOCK

// ---- FBs_Robots/FB_Joint.TcPOU
FUNCTION_BLOCK FB_Joint
VAR_INPUT
END_VAR
VAR_OUTPUT
END_VAR
VAR
	// motor IO
	m_motorInputs AT%I*	:ST_MotorInputs;
	m_motorOutputs AT%Q* :ST_MotorOutputs;
	
	// calibrated link encoder data
	m_minLinkEncoder :DINT;
	m_maxLinkEncoder :DINT;
	m_caliLinkEncoder :DINT;
	m_linkEncCaliJntPos :LREAL;
	m_linkEncZeroCross :INT;
	m_initMotorEnc : DINT;
	m_multiCycles :INT;
	
	// joint position from link encoder after power on
	m_initLinkPos :LREAL;
	
	// data for link encoder multiple cycles
	m_lastLinkEncoder :DINT;
	m_linkEncCycles:INT;
	
	// device paramters
	m_motorEncoderRes :DINT;
	m_linkEncoderRes :DINT;
	m_motorReduction :LREAL;
	m_linkEncoderReduction :LREAL;
	m_trqConst :LREAL;
	m_maxCurrent :LREAL;
	m_motorDir :INT;								
	m_linkEncoderDir :INT;
	m_minJntPos: LREAL;
	m_maxJntPos: LREAL;
	
	// macro defined data for quick calculation
	m_trq2CurrentRatio:LREAL;
	m_current2TrqRatio:LREAL;
	m_linkEnc2PosRatio :LREAL;
	m_motorEnc2PosRatio :LREAL;
	
	// joint data
	m_curMotorPos :LREAL;
	m_curLinkPos :LREAL;
	m_curJntPos	:LREAL;
	m_curJntVel :LREAL;
	m_curJntTrq :	LREAL;
	m_cmdJntPos :LREAL;
	m_cmdJntVel :LREAL;
	m_cmdJntTrq :LREAL;
	m_lastJntPos :LREAL;
	
	// velocity filter
	m_jntVelLpf :FB_LowPassFilter;
	
	// command torque filter
	m_cmdTrqLpf :FB_LowPassFilter;
	
END_VAR

METHOD PUBLIC disable : BOOL
VAR_INPUT
END_VAR
m_motorOutputs.m_controlWord:=DriverCtrlWord_INIT;
disable:=true;
END_METHOD

METHOD PUBLIC enable : BOOL
VAR_INPUT
END_VAR
IF DriverStatusWord_INIT = m_motorInputs.m_statusWord THEN
	m_motorOutputs.m_controlWord:=DriverCtrlWord_PREOP;
	enable := FALSE;
ELSIF DriverStatusWord_PREOP = m_motorInputs.m_statusWord THEN
	m_motorOutputs.m_controlWord:=DriverCtrlWord_OP;
	enable :=  FALSE;
ELSIF DriverStatusWord_OP = m_motorInputs.m_statusWord THEN
	enable :=  TRUE;
//ELSE
//	m_motorOutputs.m_controlWord:=DriverCtrlWord_INIT;
//	enable :=  FALSE;
END_IF
END_METHOD

METHOD PUBLIC init : BOOL
VAR_INPUT
	i_armIdx :INT;
	i_jntIdx :INT;
END_VAR
// hardware parameters
m_motorEncoderRes :=g_incEncoderRes[i_jntIdx];
m_linkEncoderRes :=g_absEncoderRes[i_jntIdx];
m_motorReduction :=g_motorReduction[i_jntIdx];
m_linkEncoderReduction :=g_absEncoderReduction[i_jntIdx];
m_trqConst :=g_motorTrqConst[i_jntIdx];
m_maxCurrent :=g_motorMaxCurrent[i_jntIdx];
m_motorDir :=g_motorDir[i_armIdx,i_jntIdx];								
m_linkEncoderDir :=g_asbEncoderDir[i_armIdx,i_jntIdx];
m_minJntPos	:=g_minJntPos[i_armIdx,i_jntIdx];
m_maxJntPos	:=g_maxJntPos[i_armIdx,i_jntIdx];

//link encoder calibartion data
m_minLinkEncoder :=g_minLinkEncoder[i_armIdx, i_jntIdx] - m_linkEncoderDir*g_linkEncLimitBuffer; // expand limit
m_maxLinkEncoder :=g_maxLinkEncoder[i_armIdx, i_jntIdx] + m_linkEncoderDir*g_linkEncLimitBuffer; // expand limit
m_caliLinkEncoder :=g_caliLinkEncoder[i_armIdx, i_jntIdx];
m_linkEncCaliJntPos :=g_linkEncCaliJntPos[i_armIdx, i_jntIdx];
m_linkEncZeroCross :=g_linkEncZeroCross[i_armIdx, i_jntIdx];
m_multiCycles :=g_multipleCyclesJoint[i_armIdx,i_jntIdx];

// convert cali link encoder if joint cross zero
IF 1=m_linkEncZeroCross THEN
	IF 1=m_linkEncoderDir AND m_caliLinkEncoder < m_minLinkEncoder THEN
		m_caliLinkEncoder := g_caliLinkEncoder[i_armIdx, i_jntIdx] + m_linkEncoderRes;
	ELSIF -1=m_linkEncoderDir AND m_caliLinkEncoder < m_maxLinkEncoder THEN
		m_caliLinkEncoder := g_caliLinkEncoder[i_armIdx, i_jntIdx] + m_linkEncoderRes;
	END_IF
END_IF

// macro data
m_trq2CurrentRatio:=m_motorDir * 1000.0/(m_trqConst*m_motorReduction);
m_current2TrqRatio:=m_motorDir * (m_trqConst*m_motorReduction)/1000.0;
m_linkEnc2PosRatio := 2*PI*m_linkEncoderDir/(m_linkEncoderReduction*m_linkEncoderRes);
m_motorEnc2PosRatio := 2*PI * m_motorDir/(m_motorReduction * m_motorEncoderRes);

// motor data init
m_curJntVel:=0;
m_curJntTrq :=0;
m_cmdJntVel :=0.0;
m_cmdJntTrq :=0.0;
m_jntVelLpf.init(1, g_curJntVelLpfCutoffFreq, g_armControlFreq);
m_cmdTrqLpf.init(1, g_cmdJntTrqLpfCutoffFreq, g_armControlFreq);

// driver init value
m_motorOutputs.m_controlWord:=DriverCtrlWord_INIT;
m_motorOutputs.m_opMode:=INT_TO_SINT(DriverOPMode_Pos);
m_motorOutputs.m_cmdCurrent:=0;
m_motorOutputs.m_cmdMotorEncoder:=m_motorInputs.m_motorEncoder;
END_METHOD

METHOD initJntPos : BOOL
VAR_INPUT
END_VAR
m_lastLinkEncoder :=m_motorInputs.m_linkEncoder;
m_linkEncCycles:=0;
m_curLinkPos :=linkEnc2Pos();
m_initLinkPos:=m_curLinkPos;
m_initMotorEnc :=m_motorInputs.m_motorEncoder;
m_curMotorPos:=motorEnc2Pos();
m_curJntPos := m_curMotorPos;
m_cmdJntPos :=m_curJntPos;	
m_lastJntPos :=m_curJntPos;
END_METHOD

PROPERTY initLinkPos : lreal
GET
initLinkPos:=m_initLinkPos;
END_GET
SET
m_initLinkPos:=initLinkPos;
END_SET
END_PROPERTY

METHOD isEnabled : BOOL
VAR_INPUT
END_VAR
isEnabled :=(DriverStatusWord_OP = m_motorInputs.m_statusWord);
END_METHOD

PROPERTY jntPos : LREAL
GET
jntPos := m_curJntPos;
END_GET
END_PROPERTY

PROPERTY jntTrq : LREAL
GET
jntTrq:=m_curJntTrq;
END_GET
END_PROPERTY

PROPERTY jntVel : LREAL
GET
jntVel := m_curJntVel;
END_GET
END_PROPERTY

METHOD PROTECTED linkEnc2Pos : LREAL
VAR_INPUT
END_VAR
VAR
	incLinkPos :LREAL;
	newLinkEnc :DINT;
END_VAR
// cycle check
IF 1=m_multiCycles THEN
	IF (m_motorInputs.m_linkEncoder - m_lastLinkEncoder)*m_linkEncoderDir < -m_linkEncoderRes/2 THEN
		m_linkEncCycles :=m_linkEncCycles+1;
	ELSIF (m_motorInputs.m_linkEncoder - m_lastLinkEncoder)*m_linkEncoderDir > m_linkEncoderRes/2 THEN
		m_linkEncCycles :=m_linkEncCycles-1;
	END_IF
END_IF
m_lastLinkEncoder:=m_motorInputs.m_linkEncoder;

// convert link encoder if joint cross zero
newLinkEnc := m_motorInputs.m_linkEncoder;
IF 1=m_linkEncZeroCross AND 0 = m_multiCycles THEN
	IF 1=m_linkEncoderDir AND m_motorInputs.m_linkEncoder < m_minLinkEncoder THEN
		newLinkEnc := m_motorInputs.m_linkEncoder + m_linkEncoderRes;
	ELSIF -1=m_linkEncoderDir AND m_motorInputs.m_linkEncoder < m_maxLinkEncoder THEN
		newLinkEnc := m_motorInputs.m_linkEncoder + m_linkEncoderRes;
	END_IF
END_IF

// motion from calibrated points
incLinkPos := (newLinkEnc-m_caliLinkEncoder)*m_linkEnc2PosRatio;

// absolute joint position
linkEnc2Pos := incLinkPos + m_linkEncCaliJntPos + 2*PI* m_linkEncCycles;
END_METHOD

PROPERTY PUBLIC linkPos : LREAL
GET
linkPos:=m_curLinkPos;
END_GET
END_PROPERTY

METHOD PUBLIC motorEnc2Pos : LREAL
VAR_INPUT
END_VAR
motorEnc2Pos:= (m_motorInputs.m_motorEncoder-m_initMotorEnc)* m_motorEnc2PosRatio +m_initLinkPos;
END_METHOD

PROPERTY PUBLIC motorPos : LREAL
GET
motorPos := m_curMotorPos;
END_GET
END_PROPERTY

METHOD PROTECTED motorPos2Enc : DINT
VAR_INPUT
	i_jntPos :LREAL;
END_VAR

VAR
END_VAR
motorPos2Enc := LREAL_TO_DINT((i_jntPos-m_initLinkPos)/m_motorEnc2PosRatio + m_initMotorEnc);
END_METHOD

METHOD PUBLIC updateCmds : BOOL
VAR_INPUT
	i_opMode : E_DriverOPMode;
	i_cmdPos :LREAL;
	i_cmdTrq :LREAL;
END_VAR
m_motorOutputs.m_opMode:=INT_TO_SINT( i_opMode);
// pos mode
IF i_opMode = DriverOPMode_Pos THEN
	m_motorOutputs.m_cmdCurrent:=0;
	i_cmdPos:=LIMIT(m_minJntPos, i_cmdPos, m_maxJntPos);
	m_motorOutputs.m_cmdMotorEncoder :=motorPos2Enc(i_cmdPos);
ELSIF i_opMode = DriverOPMode_Trq THEN
	m_motorOutputs.m_cmdCurrent:=LREAL_TO_DINT(LIMIT(-m_maxCurrent, i_cmdTrq*m_trq2CurrentRatio,m_maxCurrent));
	m_motorOutputs.m_cmdMotorEncoder :=m_motorInputs.m_motorEncoder; 
END_IF
END_METHOD

METHOD PUBLIC updateStatus : BOOL
VAR_INPUT
END_VAR
// compute joint position
m_curLinkPos:= linkEnc2Pos();
m_curMotorPos:=motorEnc2Pos();
m_curJntPos := m_curMotorPos;

// compute joint velocity
m_curJntVel:= (m_curJntPos-m_lastJntPos)/g_armControlLoopInterval;
m_curJntVel := m_jntVelLpf.run(m_curJntVel);
m_lastJntPos :=m_curJntPos;

m_curJntTrq := m_motorInputs.m_current * m_current2TrqRatio;
END_METHOD

END_FUNCTION_BLOCK

// ---- FBs_BasicControllers/FB_PID.TcPOU
FUNCTION_BLOCK FB_PID
VAR_INPUT
END_VAR
VAR_OUTPUT
END_VAR
VAR
	// control parameters
	m_kp:LREAL :=0.0;
	m_kd:LREAL :=0.0;
	m_ki:LREAL :=0.0;
	m_integral:LREAL :=0.0;
	m_kiLimit:LREAL :=0.0;
	m_ctrlLimit:LREAL :=0.0;
	m_cycleTime:LREAL :=0.0;
	m_outPut:LREAL:=0;
	
	// error
	m_err:LREAL:=0;
	m_dErr:LREAL:=0;
END_VAR

METHOD init : BOOL
VAR_INPUT
	// control parameters
	i_cycleTime:LREAL :=0.0;
	i_kp:LREAL :=0.0;
	i_kd:LREAL :=0.0;
	i_ki:LREAL :=0.0;
	i_kiLimit:LREAL :=0.0;
	i_ctrlLimit:LREAL :=0.0;

END_VAR
m_kp:=i_kp;
m_kd :=i_kd;
m_ki :=i_ki;
m_integral :=0.0;
m_err:=0;
m_dErr:=0;
m_kiLimit :=i_kiLimit;
m_ctrlLimit :=i_ctrlLimit;
m_cycleTime :=i_cycleTime;
END_METHOD

METHOD PUBLIC reset : BOOL
VAR_INPUT
END_VAR
m_integral :=0.0;
m_err:=0;
m_dErr:=0;
END_METHOD

METHOD run : LREAL
VAR_INPUT
	// command value
	i_cmdQ:LREAL:=0;
	
	// current value
	i_curQ:LREAL:=0;
	
	// command derivate value
	i_cmdDq:LREAL:=0;
	
	// current derivate value
	i_curDq:LREAL:=0;
END_VAR
m_err := i_cmdQ-i_curQ;
m_dErr := i_cmdDQ-i_curDq;

// integral
m_integral := m_integral + m_ki * m_err * m_cycleTime;
m_integral := LIMIT(-m_kiLimit, m_integral, m_kiLimit);

// total output
m_outPut :=m_kp*m_err+m_kd*m_dErr + m_integral;
run:=LIMIT(-m_ctrlLimit, m_outPut, m_ctrlLimit);
END_METHOD

END_FUNCTION_BLOCK

// ---- FBs_StateControllers/FB_ArmError.TcPOU
// Brief: Master Arm Initialization
FUNCTION_BLOCK PUBLIC FB_ArmError EXTENDS FB_MasterArmCtrlBase
VAR_INPUT
END_VAR
VAR_OUTPUT
END_VAR
VAR
END_VAR

END_FUNCTION_BLOCK

// ---- FBs_StateControllers/FB_MasterArmCtrlBase.TcPOU
FUNCTION_BLOCK FB_MasterArmCtrlBase IMPLEMENTS I_MasterArmCtrl
VAR_INPUT
END_VAR
VAR_OUTPUT
END_VAR
VAR
	// flag if enter controller for the first time
	m_firstIn:BOOL:=TRUE;
	
	// flag if the controller has finished all its jobs
	m_isFinished:BOOL:=FALSE;
	
	// controller execute time period
	m_timePeriod :LREAL:=0;
	
	// arm control data
	m_cmdJntPos : VEC7d;
	m_cmdJntVel : VEC7d;
	m_cmdJntAcc : VEC7d;
	m_cmdJntTrq : VEC7d;
	m_jntOPMode : Vec7i;
	m_jntEnableFlag :Vec7i;
	m_cmdCartPose : ST_Frame;
	m_cmdCartTwist : Vec6d;
END_VAR

// override this function in each exact controller
METHOD PROTECTED calcCmdJntPos : BOOL
VAR_INPUT
	monitorAngle :LREAL;
	slaveIdx :INT;
END_VAR

VAR_IN_OUT CONSTANT
	i_masterArm :FB_MasterArm;
	i_slaveStatus :ST_SlaveStatus;
END_VAR
END_METHOD

// override this function in each exact controller
METHOD PROTECTED calcCmdJntTrq : BOOL
VAR_input
	monitorAngle :LREAL;
	slaveIdx :INT;
END_VAR

VAR_IN_OUT CONSTANT
	i_masterArm :FB_MasterArm;
	i_slaveStatus :ST_SlaveStatus;
END_VAR
// set joint torque to zero in default
m_cmdJntTrq := g_zeroVec7d;
END_METHOD

// override this function in each exact controller
// NOTICE: set joint control mode here, and do some initialization if needed
METHOD PROTECTED Init : BOOL
VAR_IN_OUT CONSTANT
	i_masterArm	:FB_MasterArm;
	i_masterArmCtrlCmd :ST_ArmCtrlCmds;
END_VAR
VAR
	i:INT;
END_VAR
m_timePeriod:=0;
m_jntEnableFlag :=g_onesVec7i;
m_jntOPMode:=g_allPosMode;
m_cmdCartPose:=i_masterArm.curCartPose;
m_cmdCartTwist:=g_zeroVec6d;
m_cmdJntPos:=i_masterArm.curJntPos;
m_cmdJntVel:=g_zeroVec7d;
m_cmdJntAcc:=g_zeroVec7d;
m_cmdJntTrq:=g_zeroVec7d;
END_METHOD

PROPERTY isFinished : BOOL
GET
isFinished:=m_isFinished;
END_GET
END_PROPERTY

{warning '添加方法实现'}
METHOD reset : BOOL
m_firstIn:=TRUE;
m_isFinished:=FALSE;
END_METHOD

{warning '添加方法实现'}
METHOD run : BOOL
VAR_INPUT
	monitorAngle :LREAL;
	slaveIdx :INT;
END_VAR

VAR_IN_OUT CONSTANT
	i_masterArm :FB_MasterArm;
	i_slaveStatus :ST_SlaveStatus;
END_VAR
VAR_IN_OUT
	r_masterArmCtrlCmd :ST_ArmCtrlCmds;
END_VAR
VAR
	i:INT;
END_VAR
IF m_firstIn THEN
	Init(i_masterArm,r_masterArmCtrlCmd);
	m_firstIn:=FALSE;
END_IF

// check if arm enabled
IF FALSE = i_masterArm.isEnabled(m_jntEnableFlag) THEN
//	RETURN;
END_IF

// calculate command joint position--Motion control
calcCmdJntPos(monitorAngle, slaveIdx, i_masterArm,i_slaveStatus);

// calculate command joint torque -- Force control
calcCmdJntTrq(monitorAngle, slaveIdx, i_masterArm,i_slaveStatus);

// update commands to arm
r_masterArmCtrlCmd.m_jntEnableFlag :=m_jntEnableFlag;
r_masterArmCtrlCmd.m_cmdCartPose:=m_cmdCartPose;
r_masterArmCtrlCmd.m_cmdCartTwist:=m_cmdCartTwist;
r_masterArmCtrlCmd.m_cmdJntPos:=m_cmdJntPos;
r_masterArmCtrlCmd.m_cmdJntVel:=m_cmdJntVel;
r_masterArmCtrlCmd.m_cmdJntAcc:=m_cmdJntAcc;
r_masterArmCtrlCmd.m_cmdJntTrq:=m_cmdJntTrq;
r_masterArmCtrlCmd.m_jntOPMode:=m_jntOPMode;

// update time period
m_timePeriod := m_timePeriod+g_armControlLoopInterval;
END_METHOD

END_FUNCTION_BLOCK

// ---- FBs_StateControllers/FB_ArmInit.TcPOU
// Brief: Master Arm Initialization
FUNCTION_BLOCK PUBLIC FB_ArmInit EXTENDS FB_MasterArmCtrlBase
VAR_INPUT
END_VAR
VAR_OUTPUT
END_VAR
VAR
	m_jnt7SelfCheckVel : LREAL :=90*g_deg2Rad;
	m_jnt7HalfMotionRange : LREAL := 1.75*PI+0.26;
	m_jnt7LimitErr :LREAL := 5*g_deg2Rad;
	m_jnt7CenterPos :LREAL;
	// 0: driver on; 1: joint 7 move to upper limit, 2: joint 7 mvoe to center
	m_initState :INT :=0;
END_VAR

// override this function in each exact controller
METHOD PROTECTED calcCmdJntPos : BOOL
VAR_INPUT
	monitorAngle :LREAL;
	slaveIdx :INT;
END_VAR

VAR_IN_OUT CONSTANT
	i_masterArm :FB_MasterArm;
	i_slaveStatus :ST_SlaveStatus;
END_VAR

VAR
	centerVel:LREAL;
	curJntPos:Vec7d;
END_VAR
IF m_isFinished THEN
	RETURN;
END_IF

curJntPos :=i_masterArm.curJntPos;
CASE m_initState OF
	0:
		m_cmdJntPos := i_masterArm.curJntPos;
		IF i_masterArm.isEnabled(m_jntEnableFlag) = TRUE THEN
			m_initState :=1;
		END_IF
	1: 
		m_cmdJntPos[7] := m_cmdJntPos[7] + m_jnt7SelfCheckVel * g_armControlLoopInterval;
		IF m_cmdJntPos[7]-curJntPos[7] > m_jnt7LimitErr THEN
			m_cmdJntPos[7]:=curJntPos[7];
			m_jnt7CenterPos :=m_cmdJntPos[7]-m_jnt7HalfMotionRange;
			m_initState :=2;
		END_IF
	2:
		centerVel :=LIMIT(-m_jnt7SelfCheckVel,(m_jnt7CenterPos-m_cmdJntPos[7])/g_armControlLoopInterval,m_jnt7SelfCheckVel);
		m_cmdJntPos[7] := m_cmdJntPos[7] + centerVel * g_armControlLoopInterval;
		IF ABS(m_jnt7CenterPos-curJntPos[7]) < g_jntCtrlPosTol THEN
			m_isFinished :=TRUE;
		END_IF
END_CASE
END_METHOD

// override this function in each exact controller
// NOTICE: set joint control mode here, and do some initialization if needed
METHOD PROTECTED Init : BOOL
VAR_IN_OUT CONSTANT
	i_masterArm	:FB_MasterArm;
	i_masterArmCtrlCmd :ST_ArmCtrlCmds;
END_VAR
VAR
	i:INT;
END_VAR
SUPER^.Init(i_masterArm,i_masterArmCtrlCmd);
m_initState :=0;
END_METHOD

END_FUNCTION_BLOCK

// ---- FBs_StateControllers/FB_ArmHome.TcPOU
// Brief: Master Arm Initialization
FUNCTION_BLOCK PUBLIC FB_ArmHome EXTENDS FB_MasterArmCtrlBase
VAR_INPUT
END_VAR
VAR_OUTPUT
END_VAR
VAR
	m_homePlanner : FB_TrajMoveJ;
	
END_VAR

// override this function in each exact controller
METHOD PROTECTED calcCmdJntPos : BOOL
VAR_INPUT
	monitorAngle :LREAL;
	slaveIdx :INT;
END_VAR

VAR_IN_OUT CONSTANT
	i_masterArm :FB_MasterArm;
	i_slaveStatus :ST_SlaveStatus;
END_VAR
VAR 
	i :INT;
	curJntVel :Vec7d;
END_VAR
// check if planner is ready
IF m_homePlanner.isGene = FALSE THEN
	calcCmdJntPos:=FALSE;
	RETURN;
END_IF

// traj plan
calcCmdJntPos :=m_homePlanner.evaluate(m_timePeriod, m_cmdJntPos,m_cmdJntVel, m_cmdJntAcc);

// check if to terminate
curJntVel :=i_masterArm.curJntVel;
m_isFinished :=m_timePeriod > m_homePlanner.duration  AND normVec7(curJntVel)<7*g_jntStaticVelThres;
END_METHOD

// override this function in each exact controller
// NOTICE: set joint control mode here, and do some initialization if needed
METHOD PROTECTED Init : BOOL
VAR_IN_OUT CONSTANT
	i_masterArm :FB_MasterArm;
	i_masterArmCtrlCmd :ST_ArmCtrlCmds;
END_VAR
VAR
	i,j :INT;
	homePosture:ARRAY[1..2] OF Vec7d;
	startJntPos,endJntPos :Vec7d;
END_VAR
SUPER^.Init(i_masterArm,i_masterArmCtrlCmd);

// traj plan
startJntPos:=i_masterArm.curJntPos;
FOR j:=1 TO 7 DO 
endJntPos[j]:=g_homePosture[i_masterArm.armIdx,j];
END_FOR
m_homePlanner.init(startJntPos,endJntPos,g_homeMaxjntVel,g_homeMaxjntAcc,g_homeMaxjntJerk);
END_METHOD

END_FUNCTION_BLOCK

// ---- FBs_TrajectoryPlanning/FB_TrajMoveJ.TcPOU
FUNCTION_BLOCK FB_TrajMoveJ EXTENDS FB_TrajBase
VAR_OUTPUT
END_VAR
VAR
	// move vector in joint space
	m_startPos:Vec7d;
	m_targetPos:Vec7d;
	m_moveDir : Vec7d;
	m_moveDistance :LREAL;
	
	// doubleS planning for move distance
	m_doubleS :FB_BasicDoubleS;
END_VAR

METHOD evaluate : BOOL
VAR_INPUT
	t :LREAL;
END_VAR

VAR_IN_OUT
	jntPos,jntVel, jntAcc :vec7d;
END_VAR
VAR
	q,q_dot,q_ddot :LREAL;
END_VAR
evaluate:=m_doubleS.evaluate(t,q=>q,q_dot=>q_dot, q_ddot=>q_dot);
IF evaluate =FALSE THEN
	RETURN;
END_IF

jntPos := multiNumVec7(q, m_moveDir);
jntPos:=addVec7(jntPos, m_startPos);
jntVel := multiNumVec7(q_dot, m_moveDir);
jntAcc := multiNumVec7(q_ddot, m_moveDir);
END_METHOD

METHOD init : BOOL
VAR_IN_OUT CONSTANT
	i_startJntPos :Vec7d;
	i_targetJntPos :Vec7d;
	i_maxJntVel : Vec7d;
	i_maxJntAcc : Vec7d;
	i_maxJntJerk :Vec7d;
END_VAR
VAR 
	i:INT;
	maxV, maxA, maxJ :LREAL;
	q:ARRAY[1..2] OF LREAL;
	v:ARRAY[1..2] OF LREAL;
END_VAR
m_startPos:=i_startJntPos;
m_targetPos:=i_targetJntPos;
m_moveDir:=subVec7(i_targetJntPos, i_startJntPos);
m_moveDistance := normVec7(m_moveDir);

IF(m_moveDistance<g_smallNum) THEN
	m_moveDir:=multiNumVec7(1/7, g_onesVec7d);;
ELSE
	m_moveDir:=multiNumVec7(1/m_moveDistance, m_moveDir);
END_IF

// determian max vel/acc/jerk
maxV:=g_largeNum;
maxA:=g_largeNum;
maxJ:=g_largeNum;
FOR i :=1 TO 7 DO 
	IF ABS(m_moveDir[i])>g_smallNum THEN
		maxV := MIN (maxV, ABS(i_maxJntVel[i]/m_moveDir[i]));
		maxA := MIN (maxA, ABS(i_maxJntAcc[i]/m_moveDir[i]));
		maxJ := MIN (maxJ, ABS(i_maxJntJerk[i]/m_moveDir[i]));
	END_IF
END_FOR

// planning for moving distance
q[1]:=0;
q[2]:=m_moveDistance;
v[1]:=0;
v[2]:=0;
m_doubleS.init(q,v, maxV, maxA, maxJ);
m_duration:=m_doubleS.duration;
m_isGenerated:=m_doubleS.isGene;
END_METHOD

END_FUNCTION_BLOCK

// ---- FBs_TrajectoryPlanning/FB_BasicDoubleS.TcPOU
// reference: Trajectory planning for automation machines and robots
FUNCTION_BLOCK FB_BasicDoubleS EXTENDS FB_trajBase
VAR_INPUT
END_VAR
VAR_OUTPUT
END_VAR
VAR
	// endpoints position AND velocity
	m_q :ARRAY[1..2] OF LREAL;
	m_v :ARRAY[1..2] OF LREAL;
	
	// traj constraint
	m_maxV :LREAL:=0;
	m_maxA :LREAL:=0;
	m_maxJ :LREAL:=0;
	
	// acceleration duration
	m_Taj :LREAL :=0;
	m_Ta :LREAL :=0;
	
	// constant velocity duration
	m_Tv :LREAL :=0;
	
	// deceleration duration
	m_Tdj :LREAL :=0;
	m_Td:LREAL :=0;
	
	// traj sign
	m_sign : LREAL :=1;
	
	// trajectory parmaters
	m_limitAcc :LREAL :=0;
	m_limitDec :LREAL :=0;
	m_limitVel :LREAL :=0;
END_VAR

METHOD PUBLIC evaluate : BOOL
VAR_INPUT
	t :LREAL;
END_VAR

VAR_OUTPUT
	q,q_dot,q_ddot :LREAL;
END_VAR
VAR
	q0,q1,v0,v1:LREAL;
END_VAR
IF FALSE = m_isGenerated THEN
	evaluate := FALSE;
	RETURN;
END_IF

q:=0;
q_dot:=0;
q_ddot:=0;
q0:=m_q[1];
q1:=m_q[2];
v0:=m_v[1];
v1:=m_v[2];

IF t<=0 THEN
	q:=q0;
	q_dot:=v0;
	q_ddot:=0;
ELSIF m_Taj>0 AND  t<=m_Taj THEN
	q:=q0+v0*t+m_maxJ*EXPT(t,3)/6;
	q_dot:=v0+m_maxJ*EXPT(t,2)/2;
	q_ddot:=m_maxJ*t;
ELSIF m_Ta>2*m_Taj AND  t<=m_Ta-m_Taj THEN
	q:=q0+v0*t+m_limitAcc*(3*EXPT(t,2)-3*m_Taj*t+EXPT(m_Taj,2))/6;
	q_dot:=v0+m_limitAcc*(t-m_Taj/2);
	q_ddot:=m_limitAcc;
ELSIF m_Taj>0 AND  t<=m_Ta THEN
	q:=q0+(v0+m_limitVel)*m_Ta/2-m_limitVel*(m_Ta-t)+m_maxJ*EXPT(m_Ta-t,3)/6;
	q_dot:=m_limitVel-m_maxJ*EXPT(m_Ta-t,2)/2;
	q_ddot:=m_maxJ*(m_Ta-t);
ELSIF m_Tv>0 AND  t<=m_Ta+m_Tv THEN
	q:=q0+(v0+m_limitVel)*m_Ta/2+m_limitVel*(t-m_Ta);
	q_dot:=m_limitVel;
	q_ddot:=0;
ELSIF m_Tdj>0 AND  t<=m_Ta+m_Tv+m_Tdj THEN
	q:=q1-(m_limitVel+v1)*m_Td/2+m_limitVel*(t-m_duration+m_Td)-m_maxJ*EXPT(t-m_duration+m_Td,3)/6;
	q_dot:=m_limitVel-m_maxJ*EXPT(t-m_duration+m_Td,2)/2;
	q_ddot:=-m_maxJ*(t-m_duration+m_Td);
ELSIF m_Td>2*m_Tdj AND  t<=m_duration-m_Tdj THEN
	q:=q1-(m_limitVel+v1)*m_Td/2+m_limitVel*(t-m_duration+m_Td)+m_limitDec*(3*expt(t-m_duration+m_Td,2)-3*m_Tdj*(t-m_duration+m_Td)+m_Tdj*m_Tdj)/6;
	q_dot:=m_limitVel+m_limitDec*(t-m_duration+m_Td-m_Tdj/2);
	q_ddot:=m_limitDec;
ELSIF m_Tdj>0 AND  t<=m_duration THEN
	q:=q1-v1*(m_duration-t)-m_maxJ*EXPT(m_duration-t,3)/6;
	q_dot:=v1+m_maxJ*EXPT(m_duration-t,2)/2;
	q_ddot:=-m_maxJ*(m_duration-t);
ELSIF t>m_duration THEN
	q:=q1;
	q_dot:=v1;
	q_ddot:=0;
END_IF

q:=m_sign*q;
q_dot:=m_sign*q_dot;
q_ddot:=m_sign*q_dot;
evaluate := TRUE;
END_METHOD

METHOD PUBLIC init : BOOL
VAR_INPUT
	q :ARRAY[1..2] OF LREAL;
	v :ARRAY[1..2] OF LREAL;
	maxV :LREAL;
	maxA :LREAL;
	maxJ :LREAL;
END_VAR
VAR
	q0,q1,v0,v1,h,Delta :LREAL;
	recursiveStep :LREAL :=0.8;
	maxRecursiveTime :INT :=10;
	recursiveTime :INT :=0;
END_VAR
//normalize computation AND parameters
m_isGenerated:=FALSE;
IF q[2]=q[1] THEN
	m_sign:=1;
else
	m_sign:=(q[2]-q[1])/ABS(q[2]-q[1]);
END_IF
m_q[1]:=m_sign*q[1];
m_q[2]:=m_sign*q[2];
m_v[1]:=m_sign*v[1];
m_v[2]:=m_sign*v[2];
m_maxV:=maxV;
m_maxA:=maxA;
m_maxJ:=maxJ;

// set initial and final parameters
q0:=m_q[1];
q1:=m_q[2];
v0:=m_v[1];
v1:=m_v[2];
h:=q1-q0;

// check if traj is feasible
IF trajCheck(q1-q0,v0,v1,maxA,maxJ)=FALSE THEN 
	init :=FALSE;
	RETURN;
END_IF

// if initial and final position is same
IF ABS(q1-q0)<g_smallNum THEN
	m_Tv:=g_smallNum;
	m_duration:=g_smallNum;
	m_isGenerated:=TRUE;
	return;
END_IF

// assuming tha maxV are reached and compute the time intervel of constant velocity
// maxA not reached
IF maxA*maxA>(maxV-v0)*maxJ THEN
	m_Taj:=SQRT((maxV-v0)/maxJ);
	m_Ta:=2*m_Taj;
	m_limitAcc:=m_Taj*maxJ;
// maxA reached
else
	m_Taj:=maxA/maxJ;
	m_Ta:=m_Taj+(maxV-v0)/maxA;
	m_limitAcc:=maxA;
END_IF

// minA not reached
IF maxA*maxA>(maxV-v1)*maxJ THEN
	m_Tdj:=SQRT((maxV-v1)/maxJ);
	m_Td:=2*m_Tdj;
	m_limitDec:=-m_Tdj*maxJ;
// minA reached
else
	m_Tdj:=maxA/maxJ;
	m_Td:=m_Tdj+(maxV-v1)/maxA;
	m_limitDec:=-maxA;
END_IF
m_Tv:=(q1-q0)/maxV-m_Ta*(1+v0/maxV)/2-m_Td*(1+v1/maxV)/2;

// maxV reached
IF m_Tv>0 THEN
	m_limitVel:=maxV;
	m_isGenerated:=TRUE;
// maxV not reached, in this case, maxA must reach
else
	m_Tv:=0;
	recursiveTime:=0;
	WHILE(m_isGenerated=FALSE AND recursiveTime<maxRecursiveTime) DO
		m_Taj:=maxA/maxJ;
		m_Tdj:=maxA/maxJ;
		Delta:=EXPT(maxA,4)/EXPT(maxJ,2)+2*(v0*v0+v0*v1)+maxA*(4*h-2*maxA*(v0+v1)/maxJ);
		m_Ta:=(maxA*maxA/maxJ-2*v0+SQRT(Delta))/(2*maxA);
		m_Td:=(maxA*maxA/maxJ-2*v1+SQRT(Delta))/(2*maxA);
		IF(m_Ta<0 AND v0>v1) THEN
			m_Taj:=0;
			m_Ta:=0;
			m_Td:=2*h/(v1+v0);
			m_Tdj:=(maxJ*h-SQRT(maxJ*(maxJ*h*h+EXPT(v0+v1,2)*(v1-v0))))/(maxJ*(v1+v0));
			m_isGenerated:=TRUE;
		ELSIF(m_Td<0 AND v1>v0) THEN
			m_Tdj:=0;
			m_Td:=0;
			m_Ta:=2*h/(v1+v0);
			m_Taj:=(maxJ*h-SQRT(maxJ*(maxJ*h*h-EXPT(v0+v1,2)*(v1-v0))))/(maxJ*(v1+v0));
			m_isGenerated:=TRUE;
		END_IF

		IF m_Ta>=2*m_Taj AND m_Td>=2*m_Tdj THEN
			m_isGenerated:=TRUE;
		END_IF

		IF m_isGenerated=TRUE THEN
			m_limitAcc:=maxJ*m_Taj;
			m_limitDec:=-maxJ*m_Tdj;
			m_limitVel:=v0+(m_Ta-m_Taj)*m_limitAcc;
			RETURN;       
		END_IF
		recursiveTime:=recursiveTime+1;
		maxA:=maxA*recursiveStep;
	END_WHILE
END_IF

// total duration
m_duration:=m_Ta+m_Tv+m_Td;
m_isGenerated:=TRUE;
END_METHOD

// check if the trajectory is feasible
METHOD PROTECTED trajCheck : BOOL
VAR_INPUT
	h : LREAL;
	v0 : LREAL;
	v1 : LREAL;
	maxA : LREAL;
	maxJ : LREAL;
END_VAR
VAR
	T1,T2,dis,t :LREAL;
END_VAR
T1:=SQRT(ABS(v1-v0)/maxJ);
T2:=maxA/maxJ;
t:=MIN(T1,T2);
IF t<T2 THEN
	dis:=t*ABS(v0+v1);
else
	dis:=ABS(v0+v1)*(t+ABS(v1-v0)/maxA)/2;
END_IF

IF ABS(h)>=dis THEN 
	trajCheck:=TRUE;
else
	trajCheck:=FALSE;
END_IF
END_METHOD

END_FUNCTION_BLOCK

// ---- AgiMaths/multiNumVec7.TcPOU
FUNCTION multiNumVec7 : Vec7d
VAR_INPUT
	i_num :LREAL;
END_VAR
VAR_IN_OUT CONSTANT
	i_vec:Vec7d;
END_VAR
VAR
	i: INT ;
END_VAR

FOR i:=1 TO 7 DO 
	multiNumVec7[i]:=i_vec[i]*i_num;
END_FOR

END_FUNCTION

// ---- AgiMaths/normVec7.TcPOU
FUNCTION normVec7 : LREAL
VAR_IN_OUT CONSTANT
	vec7 :Vec7d;
END_VAR
VAR
	i:INT;
END_VAR

normVec7:=SQRT(vec7[1]*vec7[1]+vec7[2]*vec7[2]+vec7[3]*vec7[3] + 
				vec7[4]*vec7[4]+vec7[5]*vec7[5]+vec7[6]*vec7[6]+vec7[7]*vec7[7]);

END_FUNCTION

// ---- FBs_StateControllers/FB_ArmStandBy.TcPOU
// Brief: Master Arm Initialization
FUNCTION_BLOCK PUBLIC FB_ArmStandBy EXTENDS FB_MasterArmCtrlBase
VAR_INPUT
END_VAR
VAR_OUTPUT
END_VAR
VAR
END_VAR

// override this function in each exact controller
// NOTICE: set joint control mode here, and do some initialization if needed
METHOD PROTECTED Init : BOOL
VAR_IN_OUT CONSTANT
	i_masterArm :FB_MasterArm;
	i_masterArmCtrlCmd :ST_ArmCtrlCmds;
END_VAR
VAR
	j:INT;
	maxJntErr:LREAL;
	jntCtrlErr:Vec7d;
END_VAR
SUPER^.Init(i_masterArm,i_masterArmCtrlCmd);

// check if to hold the command joint position unchanged
jntCtrlErr:=subVec7(i_masterArmCtrlCmd.m_cmdJntPos, i_masterArm.m_curJntPos);
maxJntErr:=0.0;
FOR j:=1 TO g_mJntNum DO
	maxJntErr:= MAX(maxJntErr, ABS(jntCtrlErr[j]));
END_FOR

IF maxJntErr<g_jntCtrlErrForCmdHold THEN
	m_cmdJntPos:=i_masterArmCtrlCmd.m_cmdJntPos;
ELSE
	m_cmdJntPos:=i_masterArm.curJntPos;
END_IF
END_METHOD

END_FUNCTION_BLOCK

// ---- FBs_StateControllers/FB_ArmMatching.TcPOU
// Brief: Master Arm Initialization
FUNCTION_BLOCK PUBLIC FB_ArmMatching EXTENDS FB_MasterArmCtrlBase
VAR_INPUT
END_VAR
VAR_OUTPUT
END_VAR
VAR
END_VAR

END_FUNCTION_BLOCK

// ---- FBs_StateControllers/FB_ArmReady.TcPOU
// Brief: Master Arm Initialization
FUNCTION_BLOCK PUBLIC FB_ArmReady EXTENDS FB_MasterArmCtrlBase
VAR_INPUT
END_VAR
VAR_OUTPUT
END_VAR
VAR
END_VAR

END_FUNCTION_BLOCK

// ---- FBs_StateControllers/FB_ArmMasterSlave.TcPOU
// Brief: Master Arm MasterSlave controller
FUNCTION_BLOCK PUBLIC FB_ArmMasterSlave EXTENDS FB_MasterArmCtrlBase
VAR_INPUT
END_VAR
VAR_OUTPUT
END_VAR
VAR
	// joint4 controller
	m_redunJntCtrl : FB_RedunJntControl;
	
	// flag if project joint4 torque to nullspace
	m_nullspaceCtrl : BOOL :=FALSE;
	

END_VAR

// override this function in each exact controller
METHOD PROTECTED calcCmdJntPos : BOOL
VAR_INPUT
	monitorAngle :LREAL;
	slaveIdx :INT;
END_VAR

VAR_IN_OUT CONSTANT
	i_masterArm :FB_MasterArm;
	i_slaveStatus :ST_SlaveStatus;
END_VAR
var 

END_VAR
m_cmdJntPos:=i_masterArm.curJntPos;
m_cmdJntVel:=i_masterArm.curJntVel;
END_METHOD

// override this function in each exact controller
METHOD PROTECTED calcCmdJntTrq : BOOL
VAR_input
	monitorAngle :LREAL;
	slaveIdx :INT;
END_VAR

VAR_IN_OUT CONSTANT
	i_masterArm :FB_MasterArm;
	i_slaveStatus :ST_SlaveStatus;
END_VAR

VAR 
	nullspaceMat :Mat7d;
	ctrlTrq : Vec7d;
END_VAR
// redundant joint4 controller
ctrlTrq := g_zeroVec7d;
ctrlTrq[4] := m_redunJntCtrl.run(i_masterArm);

// project to nullspace
IF m_nullspaceCtrl THEN
	nullspaceMat:=i_masterArm.dynaNullspace;
	matMultiVec(nullspaceMat,ctrlTrq, m_cmdJntTrq);
	vecSelfMultiNum(m_cmdJntTrq, ctrlTrq[4] / m_cmdJntTrq[4]);
//	m_cmdJntTrq[5]:=0;
//	m_cmdJntTrq[6]:=0;
//	m_cmdJntTrq[7]:=0;
ELSE
	m_cmdJntTrq := ctrlTrq;
END_IF
END_METHOD

// override this function in each exact controller
// NOTICE: set joint control mode here, and do some initialization if needed
METHOD PROTECTED Init : BOOL
VAR_IN_OUT CONSTANT
	i_masterArm	:FB_MasterArm;
	i_masterArmCtrlCmd :ST_ArmCtrlCmds;
END_VAR
VAR
	i:INT;
END_VAR
SUPER^.Init(i_masterArm,i_masterArmCtrlCmd);

m_jntOPMode := g_allTrqMode;

// init controller
m_redunJntCtrl.init(i_masterArm);
END_METHOD

END_FUNCTION_BLOCK

// ---- MatrixLib/matMultiVec.TcPOU
// vecB = matA * vecA
FUNCTION matMultiVec : bool
VAR_IN_OUT CONSTANT
	matA :ARRAY[*,*] OF LREAL;//m*n
	vecA:ARRAY[*] OF LREAL; // n*1
END_VAR
VAR_IN_OUT 
		vecB :ARRAY[*] OF LREAL;
END_VAR
VAR
	m,n :DINT;
	i,j, k :DINT;
 
END_VAR

m:=UPPER_BOUND(matA,1);
n:= UPPER_BOUND(matA,2);
FOR i:=1 TO m DO
	vecB[i]:=0.0;
	FOR j:=1 TO n DO
		vecB[i]:=vecB[i]+matA[i,j]*vecA[j];
	END_FOR
END_FOR

END_FUNCTION

// ---- MatrixLib/vecSelfMultiNum.TcPOU
// vecA*=num
FUNCTION vecSelfMultiNum : BOOL
VAR_IN_OUT 
	vecA :ARRAY[*] OF LREAL;
END_VAR

VAR_INPUT
	num :LREAL;
END_VAR

VAR
	m :DINT;
	i :DINT;
 
END_VAR

m:=UPPER_BOUND(vecA,1);

FOR i:=1 TO m DO
		vecA[i]:=num*vecA[i];
END_FOR

END_FUNCTION

// ---- FBs_StateControllers/FB_ArmClutch.TcPOU
// Brief: Master Arm Initialization
FUNCTION_BLOCK PUBLIC FB_ArmClutch EXTENDS FB_MasterArmCtrlBase
VAR_INPUT
END_VAR
VAR_OUTPUT
END_VAR
VAR
END_VAR

END_FUNCTION_BLOCK

// ---- FBs_StateControllers/FB_ArmEndoscope.TcPOU
// Brief: Master Arm Initialization
FUNCTION_BLOCK PUBLIC FB_ArmEndoscope EXTENDS FB_MasterArmCtrlBase
VAR_INPUT
END_VAR
VAR_OUTPUT
END_VAR
VAR
END_VAR

END_FUNCTION_BLOCK

// ---- FBs_StateControllers/FB_ArmCart.TcPOU
// Brief: Master Arm Initialization
FUNCTION_BLOCK PUBLIC FB_ArmCart EXTENDS FB_MasterArmCtrlBase
VAR_INPUT
END_VAR
VAR_OUTPUT
END_VAR
VAR
END_VAR

END_FUNCTION_BLOCK

// ---- Mains/RobotDynamics.TcPOU
PROGRAM RobotDynamics

VAR
	// master robot arms joint data
	m_masterJointsData AT %I* :ST_MasterJointData;
	
	// dynamic output
	m_masterDynaData AT %Q* : ST_MasterDynaData;
	
	// flag to init robot dynamic model
	m_robotDynaInit :BOOL :=FALSE;
	
	// grivity model block
	m_gravityModel :ARRAY[1..g_mArmNum] OF FB_MasterGravity;
	
	// master arm dynamic model
	m_armDynamic :ARRAY[1..g_mArmNum] OF FB_MasterDynamic;
	
	// code execute time measure
	m_codeTime : Profiler;
	m_codeTime1 : Profiler;
	
	i: INT;
	
END_VAR

m_codeTime(START:=TRUE, RESET:=TRUE);

// robot dynamic model init
IF m_robotDynaInit =FALSE THEN
	FOR i:=1 TO g_mArmNum DO
		m_gravityModel[i].Init(i);
		m_armDynamic[i].init(i);
	END_FOR

	m_robotDynaInit:=TRUE;
END_IF

// run gravity model
FOR i:=1 TO g_mArmNum DO
	m_gravityModel[i].run(m_masterJointsData.m_curJntPos[i], m_masterDynaData.m_gravity[i]);
END_FOR

// run dynamic model
FOR i:=1 TO g_mArmNum DO
	m_armDynamic[i].updateDynamic(m_masterJointsData.m_curJntPos[i]);
	m_masterDynaData.m_massMat[i]:=m_armDynamic[i].jntMassMat;
	m_masterDynaData.m_lambda[i]:=m_armDynamic[i].cartMassMat;
	m_masterDynaData.m_dynaNullspace[i]:=m_armDynamic[i].dynaNullspace;
END_FOR

m_codeTime(START:=FALSE);

END_PROGRAM

// ---- FBs_RobotDynamics/FB_MasterGravity.TcPOU
FUNCTION_BLOCK FB_MasterGravity
VAR_INPUT
END_VAR
VAR_OUTPUT
END_VAR
VAR
	// arm index
	m_armIdx :INT;
	
	(*graParam=[ 2.7244*m3 + 2.7244*m4 + 2.7244*m5 + 2.7244*m6 + 9.8*mx2 + 9.8*mx9,
            	9.8*my2 + 9.8*my9,
			 	3.577*m4 + 3.577*m5 + 3.577*m6 + 0.49*m9 + 9.8*mx3 + 9.8*mx8
           		1.5827*m4 + 1.5827*m5 + 1.5827*m6 + 9.8*my3 + 9.8*my8 + 9.8*mz4
            	mz5-my4,	my5+mz6,  	mx4,   	mx5, 	mx6,   	my6
            	preF2,   k2,   preF3,    k3,    preF5   k5]*)
	m_gravityParam :ARRAY[1..16] OF REAL;
	// spring2 [L0, b1, b2, l1, r0]
	m_spring2Param :ARRAY[1..5] OF LREAL;
	// spring3 [L0, b1, b2, l1, r0,d]
	m_spring3Param :ARRAY[1..6] OF LREAL;
	// spring5 [L0, s1, L1, r0, beta]
	m_spring5Param :ARRAY[1..5] OF LREAL;
END_VAR

METHOD protected getRegMat : BOOL
VAR_INPUT
	// 0 for left, 1 for right
	i_armIdx:INT;
END_VAR
VAR_IN_OUT CONSTANT
	// position of all the active joint
	i_jointPos:ARRAY[1..7] OF LREAL;
END_VAR
VAR_IN_OUT
	o_regMat:ARRAY[1..5,1..16] OF LREAL;
END_VAR
VAR
	q2,q8,q4,q5,q6:LREAL;
	i,j :INT;
END_VAR
q2:=i_jointPos[2];
q8:=i_jointPos[3];
q4:=i_jointPos[4];
q5:=i_jointPos[5];
q6:=i_jointPos[6];

FOR i:=1 TO 5 DO
	FOR j:=1 TO 16 DO
		o_regMat[i,j]:=0;
	END_FOR
END_FOR

// active joint 2
o_regMat[1,1]:=COS(q2);
o_regMat[1,2]:=-SIN(q2); 
o_regMat[1,3] := 0;
o_regMat[1,4] :=   0;
o_regMat[1,5] := - 4.9*(COS(q2 - q4) - COS(q4 - q2 + 2.0*q8));
o_regMat[1,6] :=  9.8*COS(q4 - q2 + q8)*SIN(q5)*SIN(q8);
o_regMat[1,7] :=   - 4.9*(SIN(q2 - q4) + SIN(q4 - q2 + 2.0*q8));
o_regMat[1,8] :=   - 9.8*COS(q4 - q2 + q8)*COS(q5)*SIN(q8);
o_regMat[1,9] :=  9.8*SIN(q8)*(SIN(q4 - q2 + q8)*SIN(q6) - COS(q4 - q2 + q8)*COS(q5)*COS(q6));
o_regMat[1,10] :=9.8*SIN(q8)*(SIN(q4 - q2 + q8)*COS(q6) + COS(q4 - q2 + q8)*COS(q5)*SIN(q6));
spring2RegMat(q2, o_preF=>o_regMat[1,11], o_stiff=>o_regMat[1,12]);
o_regMat[1,11]:=-o_regMat[1,11];         
o_regMat[1,12]:=-o_regMat[1,12];

// active joint3
o_regMat[2,3]:= COS(q8);
o_regMat[2,4]:= - SIN(q8);
o_regMat[2,5]:= -9.8*(COS(2.0*q8)*COS(q2)*COS(q4) + COS(2.0*q8)*SIN(q2)*SIN(q4) - SIN(2.0*q8)*COS(q2)*SIN(q4) + SIN(2.0*q8)*COS(q4)*SIN(q2));
o_regMat[2,6]:= -9.8*(COS(q5)*SIN(q8) + COS(2.0*q8)*COS(q2)*SIN(q4)*SIN(q5) - COS(2.0*q8)*COS(q4)*SIN(q2)*SIN(q5) + SIN(2.0*q8)*COS(q2)*COS(q4)*SIN(q5) + SIN(2.0*q8)*SIN(q2)*SIN(q4)*SIN(q5));
o_regMat[2,7]:= 9.8*(COS(2.0*q8)*COS(q2)*SIN(q4) - COS(2.0*q8)*COS(q4)*SIN(q2) + SIN(2.0*q8)*COS(q2)*COS(q4) + SIN(2.0*q8)*SIN(q2)*SIN(q4));
o_regMat[2,8]:= 9.8*(COS(2.0*q8)*COS(q2)*COS(q5)*SIN(q4) - SIN(q5)*SIN(q8) - COS(2.0*q8)*COS(q4)*COS(q5)*SIN(q2) + SIN(2.0*q8)*COS(q2)*COS(q4)*COS(q5) + SIN(2.0*q8)*COS(q5)*SIN(q2)*SIN(q4));
o_regMat[2,9]:= 9.8*(COS(2.0*q8)*COS(q2)*COS(q4)*SIN(q6) - COS(q6)*SIN(q5)*SIN(q8) + COS(2.0*q8)*SIN(q2)*SIN(q4)*SIN(q6) - SIN(2.0*q8)*COS(q2)*SIN(q4)*SIN(q6) + SIN(2.0*q8)*COS(q4)*SIN(q2)*SIN(q6) + COS(2.0*q8)*COS(q2)*COS(q5)*COS(q6)*SIN(q4) - COS(2.0*q8)*COS(q4)*COS(q5)*COS(q6)*SIN(q2) + SIN(2.0*q8)*COS(q2)*COS(q4)*COS(q5)*COS(q6) + SIN(2.0*q8)*COS(q5)*COS(q6)*SIN(q2)*SIN(q4)); 
o_regMat[2,10]:= 9.8*(SIN(q5)*SIN(q6)*SIN(q8) + COS(2.0*q8)*COS(q2)*COS(q4)*COS(q6) + COS(2.0*q8)*COS(q6)*SIN(q2)*SIN(q4) - SIN(2.0*q8)*COS(q2)*COS(q6)*SIN(q4) + SIN(2.0*q8)*COS(q4)*COS(q6)*SIN(q2) - COS(2.0*q8)*COS(q2)*COS(q5)*SIN(q4)*SIN(q6) + COS(2.0*q8)*COS(q4)*COS(q5)*SIN(q2)*SIN(q6) - SIN(2.0*q8)*COS(q2)*COS(q4)*COS(q5)*SIN(q6) - SIN(2.0*q8)*COS(q5)*SIN(q2)*SIN(q4)*SIN(q6));
spring3RegMat(q8, o_preF=>o_regMat[2,13], o_stiff=>o_regMat[2,14]);
o_regMat[2,13]:=-o_regMat[2,13];
o_regMat[2,14]:=-o_regMat[2,14];

// active joint4
o_regMat[3,5]:= 9.8*SIN(q4 - q2 + q8)*SIN(q8);
o_regMat[3,6]:= - 9.8*COS(q4 - q2 + q8)*SIN(q5)*SIN(q8);
o_regMat[3,7]:= 9.8*COS(q4 - q2 + q8)*SIN(q8);
o_regMat[3,8]:= 9.8*COS(q4 - q2 + q8)*COS(q5)*SIN(q8);
o_regMat[3,9]:= - 9.8 *SIN(q8)*(SIN(q4 - q2 + q8)*SIN(q6) - COS(q4 - q2 + q8)*COS(q5)*COS(q6));
o_regMat[3,10]:= - 9.8*SIN(q8)*(SIN(q4 - q2 + q8)*COS(q6) + COS(q4 - q2 + q8)*COS(q5)*SIN(q6));
              
// active joint5
o_regMat[4,6]:= -9.8* (COS(q8)*SIN(q5) + SIN(q4 - q2 + q8)*COS(q5)*SIN(q8));
o_regMat[4,7]:= 0;
o_regMat[4,8]:= 9.8* (COS(q5)*COS(q8) - SIN(q4 - q2 + q8)*SIN(q5)*SIN(q8));
o_regMat[4,9]:= 9.8*COS(q6)*(COS(q5)*COS(q8) - SIN(q4 - q2 + q8)*SIN(q5)*SIN(q8));
o_regMat[4,10]:= -9.8*SIN(q6)*(COS(q5)*COS(q8) - SIN(q4 - q2 + q8)*SIN(q5)*SIN(q8));
spring5RegMat(q5, o_preF=>o_regMat[4,15], o_stiff=>o_regMat[4,16]);
o_regMat[4,15]:=-o_regMat[4,15];
o_regMat[4,16]:=-o_regMat[4,16];

// active joint5
o_regMat[5,9]:= -9.8*(COS(q8)*SIN(q5)*SIN(q6) - COS(q4 - q2 + q8)*COS(q6)*SIN(q8) + SIN(q4 - q2 + q8)*COS(q5)*SIN(q6)*SIN(q8));
o_regMat[5,10]:= -9.8*(COS(q4 - q2 + q8)*SIN(q6)*SIN(q8) + COS(q6)*COS(q8)*SIN(q5) + SIN(q4 - q2 + q8)*COS(q5)*COS(q6)*SIN(q8));
END_METHOD

METHOD PUBLIC init : BOOL
VAR_INPUT
	i_armIdx :INT;
END_VAR
VAR
	i:INT;
END_VAR
m_armIdx:=i_armIdx;

FOR i:=1 TO 16 DO
	m_gravityParam[i]:=g_gravityParam[m_armIdx, i];
END_FOR

